(* CODESYS project ILG_Std_Lib
   Company: ILLIG packaging solutions
   DefaultNamespace: ILGStdLib
   Title: ILG_Std_Lib
   Version: 0.0.0.3

Project tree, tasks and I/O mapping:
  libraries: CXA_Utilities, 2.6.2.0 (Bosch Rexroth AG); CXA_CommonTypes, 3.4.0.0 (Bosch Rexroth AG); CXA_PLCopen, 3.4.0.3 (Bosch Rexroth AG); Standard, 3.5.18.0 (System); SysDir, 3.5.17.0 (System); SysFileAsync, 3.5.19.0 (System); SysTimeCore, 3.5.17.0 (System); SysTimeRtc, 3.5.20.0 (System); SysTypes, 3.1.2.0 (System); CXA_ctrlXIO, 1.20.11.0 (Bosch Rexroth AG); CXA_Datalayer, 3.4.0.0 (Bosch Rexroth AG); CXA_DriveUtil, 2.6.0.0 (Bosch Rexroth AG); CXA_FileAsync, 2.6.0.0 (Bosch Rexroth AG); CXA_Motion, 3.4.5.2 (Bosch Rexroth AG); CXA_MotionCore_fbs, 3.3.0.0 (Bosch Rexroth AG); CXA_MotionInterface, 3.4.0.3 (Bosch Rexroth AG); CXAC_Base, 1.18.4.0 (Bosch Rexroth AG); SysFile, 3.5.17.0 (System); File Access, 3.5.17.0 (3S - Smart Software Solutions GmbH); Software Engineering, 0.0.1 (Illig packaging solutions)
  libraries: CXA_Utilities, 2.6.2.0 (Bosch Rexroth AG); CXA_CommonTypes, 3.4.0.0 (Bosch Rexroth AG); CXA_PLCopen, 3.4.0.3 (Bosch Rexroth AG); Standard, 3.5.18.0 (System); SysDir, 3.5.17.0 (System); SysFileAsync, 3.5.19.0 (System); SysTimeCore, 3.5.17.0 (System); SysTimeRtc, 3.5.20.0 (System); SysTypes, 3.1.2.0 (System); CXA_ctrlXIO, 1.20.11.0 (Bosch Rexroth AG); CXA_Datalayer, 3.4.0.0 (Bosch Rexroth AG); CXA_DriveUtil, 2.6.0.0 (Bosch Rexroth AG); CXA_FileAsync, 2.6.0.0 (Bosch Rexroth AG); CXA_Motion, 3.4.5.2 (Bosch Rexroth AG); CXA_MotionCore_fbs, 3.3.0.0 (Bosch Rexroth AG); CXA_MotionInterface, 3.4.0.3 (Bosch Rexroth AG); CXAC_Base, 1.18.4.0 (Bosch Rexroth AG); SysFile, 3.5.17.0 (System); File Access, 3.5.17.0 (3S - Smart Software Solutions GmbH)
  00000000-0000-0000-0000-000000000000|D:\EIGENE_DATEIEN\GIT\libraries\SourceLibraries\CXA\CXA_Template\HistoryCXA_Template.txt
  0.7.0.0.Sync
  0.7.0.1.Sync
  _History/
    program _History_ [ST]
    History.txt
  _Library Informations/
    function GetLibVersion [ST]
    function GetLibVersionNumber [ST]
  commdata.all
  commdata.all
  commdata.all
  commdata.all
  Constants/
    GlobalKit/
      global variables GVL_ConstantsFlexProfile
      global variables GVL_ConstantsGlobalKit
  CXA_Library_Template.Sync
  function block FB_ArrayToWord_1 [ST]
  GeneralFunctionBlocks/
    ActivateDevices/
      Datatypes/
        ActConfig/
          data type ST_AxesActConfig
          data type ST_DeviceActConfig
          data type ST_DeviceActConfigBase
          data type ST_FirmwareType
          data type ST_InlineIOActConfig
          data type ST_ProfibusIOActConfig
          data type ST_SercosIOActConfig
          data type ST_SercosIOModuleActConfig
        CmdConfig/
          AxesConfig/
            data type ST_DoubleAxisConfig
            data type ST_FunctionalPackages
          data type ST_AxesCmdConfig
          data type ST_DeviceCmdConfig
          data type ST_DeviceCmdConfigBase
          data type ST_InlineIOCmdConfig
          data type ST_PNIOCmdConfig
          data type ST_PNIOModuleCmdConfig
          data type ST_ProfibusIOCmdConfig
          data type ST_SercosIOCmdConfig
          data type ST_SercosIOModuleCmdConfig
        data type E_InlineType
        data type E_S20Type
        Error/
          data type ST_AxesConfigError
          data type ST_AxesConfigErrorFoundDrives
          data type ST_DeviceConfigError
          data type ST_DeviceConfigErrorBase
          data type ST_InlineIOConfigError
          data type ST_ProfibusIOConfigError
          data type ST_SercosIOCmdConfigError
          data type ST_SercosIOConfigError
          data type ST_SercosIOModuleConfigError
        data type ST_DirEntry
        data type ST_SercosErrorReaction
      function block FB_ActivateDevices [ST]: _M_WriteLnString, M_0ReadActConfig, M_1ConfigAxes, M_2ConfigSercosIO, M_3ConfigInlineIO, M_4ConfigProfibsIO, M_5ConfigProfinetIO, M_8WriteConfig, M_9ErrorDone, M_DelStructure, M_Execute, M_GetSafetyType, M_GetSercosAdress, M_S20TypeToString, M_TypeCodeIsRexrothIO
      global variables GVL_ActivateDevices
      interface ITF_ActivateDevices: M_Execute
    ChangeNextDiagDelay/
      function block FB_ChangeNextDiagDelay [ST]
    function block FB_ArrayToWord [ST]
    function block FB_BlockAcknowledge10 [ST]
    function block FB_BlockAcknowledge21 [ST]
    function block FB_ClockMarker [ST]
    function block FB_Convert8BitTo5BitParameter [ST]
    function block FB_IlligOperatingModes [ST]
    function block FB_IlligZaehlstern [ST]
    function block FB_ParallelSteps [ST]
    function block FB_TimeBasedClockGenerator [ST]
    function block FB_TriggerValueChange [ST]
    function block FB_ValueIsIntegerMultiple [ST]
    function block FB_VIMP [ST]
  GeneralFunctions/
    Convert/
      function F_byWordToLeftByte [ST]
      function F_DwordToStrH5 [ST]
      function F_DwordToStrH8 [ST]
      function F_dwSwapDWordWord [ST]
      function F_iAnalogOutput4To20mA [ST]
      function F_rAnalogInput0To10V [ST]
      function F_rSwapReal [ST]
      function F_rSwapRealWord [ST]
      function F_Tad [ST]
      function F_WordToStrH [ST]
    ILG_Functions/
      function F_bCamDiscCalculation [ST]
      function F_InitArray [ST]
    Math/
      function F_lrRound [ST]
      function F_lrRoundRealToLReal [ST]
      function F_rModulo [ST]
      function F_rRound [ST]
      function F_rRoundGreater [ST]
      function F_rRoundTime [ST]
  Global Variables/
  ILG_Std_Lib.Sync
  ILG_Std_Lib.Sync
  ILG_Std_Lib.Sync
  ILG_Std_Lib.Sync
  InternalFunctions/
    function FUN_WriteLnString [ST]
  MachineDoorControllerInterface.Sync
  global variables ParaCxaLibraryTemplate
  program ReadMe [ST]
  Software Engineering.Sync
  Types/
    data type ST_Split
    data type T_CamTable
    data type T_ServoAxesArray
    data type T_Tables
  UnknownLibrary1.Sync
  UnknownLibrary21.Sync
  UnknownLibrary.Sync
*)

// Types/ST_Split
TYPE ST_Split :
STRUCT
	arWords:     ARRAY [1..400] OF POINTER TO STRING[255];
END_STRUCT
END_TYPE

// Types/T_CamTable
/// Ersetzt array vom Typ: ARRAY [1..99,1..1024] OF REAL; 
{attribute 'qualified_only' := ''}
{attribute 'namespace' := 'ILGStdLib.Types'}
TYPE T_CamTable :
ARRAY[1..99, 1..1024] OF REAL;
END_TYPE

// Types/T_ServoAxesArray
/// Ersetzt array vom Type: ARRAY[1..Max_Servoachsen, 0..Max_Segmente, 0..Max_Daten_pro_Segment] OF REAL
{attribute 'qualified_only' := ''}
{attribute 'namespace' := 'ILGStdLib.Types'}
TYPE T_ServoAxesArray :
ARRAY[1..GVL_ConstantsGlobalKit.iMAX_SERVO_AXES, 0..GVL_ConstantsGlobalKit.iMAX_SEGMENTS, 0..GVL_ConstantsGlobalKit.iMAX_DATA_PER_SEGMENT] OF REAL;
END_TYPE

// Types/T_Tables
/// Ersetzt array vom Type: ARRAY [1..Max_Anzahl_Stuetzpunkte, 1..Max_Anzahl_Tabellen] OF REAL; 
{attribute 'qualified_only' := ''}
{attribute 'namespace' := 'ILGStdLib.Types'}
TYPE T_Tables :
ARRAY[1..GVL_ConstantsGlobalKit.iMAX_COUNT_OF_SUPPORT_POINTS, 1..GVL_ConstantsGlobalKit.iMAX_COUNT_OF_TABLES] OF REAL;
END_TYPE

// GeneralFunctionBlocks/ActivateDevices/Datatypes/E_InlineType
{attribute 'qualified_only' := ''}
TYPE E_InlineType :
(
	///R-IB IL 24 DI 16-PAC 
	///R-IB IL 24 DI 16
	INLINE_DI16 := 16#BE01,
	///R-IB IL 24 DI 32/HD 
	///R-IB IL 24 DI 32/HD-PAC 
	///R-IB IL 24 DI 32/HD-NPN-PAC
	INLINE_DI32 := 16#BE02,
	///R-IB IL 24 DI 4
	///R-IB IL 24 DI 4-PAC
	///R-IB IL 24 EDI 2-DES
	///R-IB IL 24 DI 16-NPN-PAC 
	INLINE_DI4_2_16 := 16#BE41,
	///R-IB IL 24 DI 8
	///R-IB IL 24 DI 8-PAC
	INLINE_DI8 := 16#BE81,
	///R-IB IL 24 DI 2
	///R-IB IL 24 DI 2-PAC
	///R-IB IL 24 DI 2-NPN-PAC
	///IB IL 24 SEG/F-D-PAC
	INLINE_DI2_SEG := 16#BEC2,
	///R-IB IL 24 DO 16
	///R-IB IL 24 DO 16-PAC
	INLINE_DO16 := 16#BD01,
	///R-IB IL 24 DO 32/HD
	///R-IB IL 24 DO 32/HD-PAC
	///R-IB IL 24 DO 32/HD-NPN-PAC
	INLINE_DO32 := 16#BD02,
	///R-IB IL 24 DO 4
	///R-IB IL 24 DO 4-PAC
	///R-IB IL 24/230 DOR 4/W
	///R-IB IL 24/230 DOR 4/W-PAC
	INLINE_DO4_DOR4 := 16#BD41,
	///R-IB IL 24 DO 8
	///R-IB IL 24 DO 8-PAC
	///R-IB IL 24 DO 8-2A
	///R-IB IL 24 DO 8-2A-PAC
	///R-IB IL 24 DO 8-NPN-PAC
	INLINE_DO8 := 16#BD81,
	///R-IB IL 24 DO 2-2A
	///R-IB IL 24 DO 2-2A-PAC
	///R-IB IL 24 DO 2-NPN-PAC
	///R-IB IL 24/230 DOR 1/W
	///R-IB IL 24/230 DOR 1/W-PAC
	INLINE_DO2_DOR1 := 16#BDC2,
	///R-IB IL AI 8/SF-PAC
	///R-IB IL AI 8/IS-PAC
	INLINE_AI8 := 16#5F02,
	///R-IB IL AI 2/SF
	///R-IB IL AI 2/SF-PAC
	///R-IB IL AI 2/SF-230-PAC
	///R-IB IL TEMP 2 RTD
	///R-IB IL TEMP 2 RTD-PAC
	///R-IB IL TEMP 2 UTH-PAC
	///R-IB IL INC-IN-PAC
	INLINE_AI2_TEMP_INC_IN := 16#7F02,
	///R-IB IL SGI 2/F-PAC
	INLINE_SGI2 := 16#DF03,
	///R-IB IL AI 4/EF-PAC
	///R-IB IL TEMP 4/8 RTD-PAC
	INLINE_AI4_TEMP := 16#DF05,
	///R-IB IL AO 2/U/BP
	///R-IB IL AO 2/U/BP-PAC
	///R-IB IL AO 2/SF-PAC
	INLINE_AO2 := 16#5B02,
	///R-IB IL AO 1/SF
	///R-IB IL AO 1/SF-PAC
	INLINE_AO1 := 16#7D01,
	///R-IB IL CNT
	///R-IB IL CNT-PAC
	///R-IB IL INC-PAC
	///R-IB IL SSI-PAC
	///R-IB IL PWM/2-PAC
	///R-IB IL TEMPCON UTH-PAC
	INLINE_CNT_SSI_INC_PWM_TEMP := 16#BF02,
	///R-IL BK DDL
	INLINE_BK_DDL := 16#BF04,
	///R-IB IL RS232-PRO-PAC
	///R-IB IL RS485/422-PRO-PAC
	INLINE_RS232_RS485 := 16#BF06,
	///RF-FLM DI 8 M8
	INLINE_FLM_DI8 := 16#B281,
	///RF-FLM DIO 8/4 M8
	INLINE_FLM_DIO8 := 16#B381
);
END_TYPE

// GeneralFunctionBlocks/ActivateDevices/Datatypes/E_S20Type
{attribute 'qualified_only' := ''}
TYPE E_S20Type :
(
	///	undefinded
	S20_UNDEFINED := 16#0,
	///	S20-S3-BK+	Buskopf			R911173318
	S20_S3_BK_PLUS := 16#4158010099990002,
	///	S20-DI-16/4					R911172532
	S20_DI_16_4 := 16#41580002000000D0,
	///	S20-DO-16/3					R911172534
	S20_DO_16_3 := 16#41580002000000D1,
	///	S20-DI-32/1					R911172533
	S20_DI_32_1 := 16#41580004000000D2,
	///	S20-DO-32/1					R911172535
	S20_DO_32_1 := 16#41580004000000D3,
	///	S20-DO-8/2-2A				R911172541
	S20_DO_8_2_2A := 16#41580001000000D5,
	///	S20-DI-16/1					R911172543
	S20_DI_16_1 := 16#41580002000000D6,
	///	S20-DO-16/1					R911172542
	S20_DO_16_1 := 16#41580002000000D7,
	///	S20-AI-8					R911172536
	S20_AI_8 := 16#41580010000000A0,
	///	S20-AI-8-RTD				R911172537
	S20_AI_8_RTD := 16#41580010000000A1,
	///	S20-AI-8-UTH				R911172545               
	S20_AI_8_UTH := 16#41580012000000A2,
	///	S20-AO-8					R911172538
	S20_AO_8 := 16#41580010000000A3,
	///	S20-CNT-INC-2/2				R911172539
	S20_CNT_INC_2_2 := 16#4158001C000000F1,
	///	S20-SSI-AO-1/1				R911172544
	S20_SSI_AO_1_1 := 16#4158100C000000F2,
	///	Test_ChM					
	Placeholder_1 := 16#4158000400000008,
	///	Test_ChM					
	Placeholder_2 := 16#41580001000000D8,
	///	Test_ChM					
	Placeholder_3 := 16#4158000100000002,
	///	S20-AI-4-I					R911173249
	S20_AI_4_I := 16#41580008000000A6,
	///	S20-AI-4-U					R911173256
	S20_AI_4_U := 16#41580008000000A5,
	///	S20-DI-64/1					R911173340
	S20_DI_64_1 := 16#41580008000000D8,
	///	S20-DI-16/1-HS				R911173344
	S20_DI_16_1_HS := 16#41580002000000DB,
	///	S20-AI-4-RTD				R911173341
	S20_AI_4_RTD := 16#41580008000000A4,
	///	S20-RS-UNI					R911173343
	S20_RS_UNI := 16#41580814000000C0,
	///	S20-DIDO-8/1				R911173745               
	S20_DIDO_8_1 := 16#41580001000000DD,
	///	S20-AO-4					R911173248
	S20_AO_4 := 16#41580008000000A7,
	///	Test_ChM
	Placeholder_4 := 16#41580002000000DC,
	///	S20-AI-4-UTH				R911173342
	S20_AI_4_UTH := 16#41580008000000A8,
	///	SSDI-8/4					R911173191
	S20_SSDI_8_4 := 16#4158000A00000F00,
	///	SSDO-8/3					R911173192
	S20_SSDO_8_3 := 16#4158000A00000F01,
	///	S20-AI6-AO2-SSI2			R911173120
	S20_AI6_AO2_SSI2 := 16#41581014000000F3,
	///	S20-INC-2					R911173559
	S20_INC_2 := 16#41581014000000F5,
	///	S20-AIAO-2					R911173743
	S20_AIAO_2 := 16#41580008000000A9,
	///	S20-DO-64/1					R911173742
	S20_DO_64_1 := 16#41580008000000DF,
	///	S20-DOR-4/2-220-AC			R911173749
	S20_DOR_4_2_220_AC := 16#4158000100000D00,
	///	S20-DI-16/4-DO-8/3-HS		R911xxxxxx
	///  S20-SSI-AO-1_1				R911172544_AA1  fehlt in Buskoppler SDDML					
	S20_DI_16_4_DO_8_3_HS := 16#41580003010000D9
) LINT;
END_TYPE

// GeneralFunctionBlocks/ActivateDevices/Datatypes/ST_DirEntry
TYPE ST_DirEntry :
STRUCT
	sEntry: STRING;
	bDirectory: BOOL;
END_STRUCT
END_TYPE

// GeneralFunctionBlocks/ActivateDevices/Datatypes/ST_SercosErrorReaction
{attribute 'qualified_only' := ''}
{attribute 'strict' := ''}
TYPE ST_SercosErrorReaction :
STRUCT
	/// C-0-0506 Bit 0 = TRUE
	bF2Error: BOOL;
	/// C-0-0506 Bit 1 = TRUE
	bF5Error: BOOL;
	/// C-0-0506 Bit 0,1 = FALSE
	bF8Error: BOOL;
	/// Switch of E00B0179
	bNoRedundancyWarning: BOOL;
	bAutoRingRecovery: BOOL;
END_STRUCT
END_TYPE

// GeneralFunctionBlocks/ActivateDevices/Datatypes/ActConfig/ST_AxesActConfig
TYPE ST_AxesActConfig EXTENDS ST_DeviceActConfigBase :
STRUCT
	/// Name of Device 
	sName: STRING;
	/// TRUE = real Axis 
	bRealAxis: BOOL;
	/// TRUE = virtual Axis 
	bVirtualAxis: BOOL;
	/// Sercos address
	iSercosAddress: INT;
	/// Firmwarestring e.g. MPH-07 
	sFirmware: STRING;
	/// SNC or NOT 
	stFunctionalPackages: ST_FunctionalPackages;
	/// Which Axis of double Axis ? 
	stDoubleAxis: ST_DoubleAxisConfig;
	/// IP of drive S-0-1020
	sIP: STRING(16);
	/// serial no of Drive
	udiSerialNo: UDINT;
	/// String of SafetyType e.g. 'L3', 'S4', etc.	
	sSafetyType: STRING(2);
END_STRUCT
END_TYPE

// GeneralFunctionBlocks/ActivateDevices/Datatypes/ActConfig/ST_DeviceActConfig
TYPE ST_DeviceActConfig :
STRUCT
	astAxes: ARRAY[1..iMAX_AXES_NUMBER] OF ST_AxesActConfig;
	astSercosIO: ARRAY[1..iMAX_SERCOS_IO] OF ST_SercosIOActConfig;
	astInlineIO: ARRAY[1..iMAX_INLINE_IO] OF ST_InlineIOActConfig;
END_STRUCT
END_TYPE

// GeneralFunctionBlocks/ActivateDevices/Datatypes/ActConfig/ST_DeviceActConfigBase
TYPE ST_DeviceActConfigBase :
STRUCT
	/// TRUE = Device is present on the bus 
	bAvailable: BOOL;
END_STRUCT
END_TYPE

// GeneralFunctionBlocks/ActivateDevices/Datatypes/ActConfig/ST_FirmwareType
TYPE ST_FirmwareType :
STRUCT
	sType: STRING;
	iVersion: INT;
	iRelease: INT;
	bTestversion: BOOL;
END_STRUCT
END_TYPE

// GeneralFunctionBlocks/ActivateDevices/Datatypes/ActConfig/ST_InlineIOActConfig
TYPE ST_InlineIOActConfig EXTENDS ST_DeviceActConfigBase :
STRUCT
	eIOType: E_InlineType;
END_STRUCT
END_TYPE

// GeneralFunctionBlocks/ActivateDevices/Datatypes/ActConfig/ST_ProfibusIOActConfig
TYPE ST_ProfibusIOActConfig EXTENDS ST_DeviceActConfigBase :
STRUCT
END_STRUCT
END_TYPE

// GeneralFunctionBlocks/ActivateDevices/Datatypes/ActConfig/ST_SercosIOActConfig
TYPE ST_SercosIOActConfig EXTENDS ST_DeviceActConfigBase :
STRUCT
	/// Name of Device (will be taken from Cmd structure)
	sName: STRING;
	/// Sercos address
	iSercosAddress: INT;
	/// R911 TypeCode 
	sTypeCode: STRING;
	uiNoOfIO_Modules: UINT;
	astIOModule: ARRAY[0..GVL_ActivateDevices.iMAX_MODULE_ON_SERCOS_IO] OF ST_SercosIOModuleActConfig;
END_STRUCT
END_TYPE

// GeneralFunctionBlocks/ActivateDevices/Datatypes/ActConfig/ST_SercosIOModuleActConfig
TYPE ST_SercosIOModuleActConfig EXTENDS ST_DeviceActConfigBase :
STRUCT
	/// IO Module Type e.g. S20_DI_16_4
	IOType: E_S20Type;
END_STRUCT
END_TYPE

// GeneralFunctionBlocks/ActivateDevices/Datatypes/CmdConfig/ST_AxesCmdConfig
TYPE ST_AxesCmdConfig EXTENDS ST_DeviceCmdConfigBase :
STRUCT
	/// TRUE = real Axis 
	bRealAxis: BOOL;
	/// TRUE = virtual Axis 
	bVirtualAxis: BOOL;
	/// Sercos address
	iSercosAddress: INT;
	/// Firmwarestring e.g. MPH-07 
	sFirmware: STRING(8);
	/// SNC or NOT 
	stFunctionalPackages: ST_FunctionalPackages;
	/// String of SafetyType e.g. 'L3', 'S4', etc.
	sSafetyType: STRING(2);
	/// 	0: active, 
	///																						1: parked,
	///																						2: deactivated, 
	///																						4: active without command value processing,
	///																						5: parked with command value calculation,
	///																						6: deactivated with command value calculation 
	///																					
	iStatus: INT;
	/// Which Axis of double Axis ? 
	stDoubleAxis: ST_DoubleAxisConfig;
END_STRUCT
END_TYPE

// GeneralFunctionBlocks/ActivateDevices/Datatypes/CmdConfig/ST_DeviceCmdConfig
TYPE ST_DeviceCmdConfig :
STRUCT
	astAxes: ARRAY[1..iMAX_AXES_NUMBER] OF ST_AxesCmdConfig;
	astSercosIO: ARRAY[1..iMAX_SERCOS_IO] OF ST_SercosIOCmdConfig;
	astInlineIO: ARRAY[1..iMAX_INLINE_IO] OF ST_InlineIOCmdConfig;
	/// [x,0].Active = PROFINET MASTER is active
	astProfibusIO: ARRAY[1..iMAX_PROFIBUS_MASTER, 0..iMAX_PROFIBUS_SLAVE] OF ST_ProfibusIOCmdConfig;
	/// [x,0].Active = Profinet Master is active	(* 2020-07-06 gt: nach Vorlage "activateDevices_14.8.XM.iwz" von Jörg Schneider *)
	astPN_IO: ARRAY[1..iMAX_PN_MASTER, 0..iMAX_PN_SLAVE] OF ST_PNIOCmdConfig;
END_STRUCT
END_TYPE

// GeneralFunctionBlocks/ActivateDevices/Datatypes/CmdConfig/ST_DeviceCmdConfigBase
TYPE ST_DeviceCmdConfigBase :
STRUCT
	/// Name of Device 
	sName: STRING(80);
	/// TRUE = Device will be activated 
	bActive: BOOL;
END_STRUCT
END_TYPE

// GeneralFunctionBlocks/ActivateDevices/Datatypes/CmdConfig/ST_InlineIOCmdConfig
TYPE ST_InlineIOCmdConfig EXTENDS ST_DeviceCmdConfigBase :
STRUCT
	///IO is configured in IndraWorks	
	bConfigured: BOOL;
	/// which IO Type is used	 	
	eIOType: E_InlineType;
END_STRUCT
END_TYPE

// GeneralFunctionBlocks/ActivateDevices/Datatypes/CmdConfig/ST_PNIOCmdConfig
TYPE ST_PNIOCmdConfig EXTENDS ST_DeviceCmdConfigBase :
STRUCT
	///Fieldbus address 	
	sPNDeviceName: STRING(80);
	astIOModule: ARRAY[0..iMAX_MODULE_ON_PN_IO] OF ST_PNIOModuleCmdConfig;
END_STRUCT
END_TYPE

// GeneralFunctionBlocks/ActivateDevices/Datatypes/CmdConfig/ST_PNIOModuleCmdConfig
TYPE ST_PNIOModuleCmdConfig EXTENDS ST_DeviceCmdConfigBase :
STRUCT
	bConfigured: BOOL;
END_STRUCT
END_TYPE

// GeneralFunctionBlocks/ActivateDevices/Datatypes/CmdConfig/ST_ProfibusIOCmdConfig
TYPE ST_ProfibusIOCmdConfig EXTENDS ST_DeviceCmdConfigBase :
STRUCT
	///Fieldbus address
	iAddress: INT;
END_STRUCT
END_TYPE

// GeneralFunctionBlocks/ActivateDevices/Datatypes/CmdConfig/ST_SercosIOCmdConfig
TYPE ST_SercosIOCmdConfig EXTENDS ST_DeviceCmdConfigBase :
STRUCT
	/// Sercos address
	iSercosAddress: INT;
	///	Firmware 				:STRING;																(* Firmwarestring *)	
	astIOModule: ARRAY[0..iMAX_MODULE_ON_SERCOS_IO] OF ST_SercosIOModuleCmdConfig;
	/// will be calculated automatically if CheckSercosIOModuleConfig = TRUE
	uiNoOfIOModules: UINT;
END_STRUCT
END_TYPE

// GeneralFunctionBlocks/ActivateDevices/Datatypes/CmdConfig/ST_SercosIOModuleCmdConfig
TYPE ST_SercosIOModuleCmdConfig EXTENDS ST_DeviceCmdConfigBase :
STRUCT
	///IO Module is configured in IndraWorks		
	bConfigured: BOOL;
	/// IO Module Type e.g. S20_DI_16_4
	eIOType: E_S20Type;
END_STRUCT
END_TYPE

// GeneralFunctionBlocks/ActivateDevices/Datatypes/Error/ST_AxesConfigError
TYPE ST_AxesConfigError EXTENDS ST_DeviceConfigErrorBase :
STRUCT
	/// TRUE = Found drive has wrong SercosAddress
	bWrongSercosAddress: BOOL;
	/// TRUE = Found drive has wrong Firmware 
	bWrongFirmware: BOOL;
	/// TRUE = Found drive has wrong Functional Package
	bWrongFunctionalPackages: BOOL;
	/// TRUE = Found drive has wrong Doubleaxis Configuration
	bWrongDoubleAxisConfiguration: BOOL;
	/// TRUE = Found drive has wrong Safety option
	bWrongSafetyType: BOOL;
	/// TRUE = Drive is configured but not found
	bDriveConfiguredAndNotFound: BOOL;
	/// TRUE = Drive is found and configured in C-0-0478 (IndraWorks), but not configured at DeviceCmdConfig
	bDriveFoundAndNotConfigured: BOOL;
	/// Sercos Address of device 			
	iSercosAddress: INT;
END_STRUCT
END_TYPE

// GeneralFunctionBlocks/ActivateDevices/Datatypes/Error/ST_AxesConfigErrorFoundDrives
TYPE ST_AxesConfigErrorFoundDrives EXTENDS ST_DeviceConfigErrorBase :
STRUCT
	/// Sercos Address of device
	iSercosAddress: INT;
END_STRUCT
END_TYPE

// GeneralFunctionBlocks/ActivateDevices/Datatypes/Error/ST_DeviceConfigError
TYPE ST_DeviceConfigError :
STRUCT
	astAxes: ARRAY[1..iMAX_AXES_NUMBER] OF ST_AxesConfigError;
	///drive which were found but not configured in C-0-0478
	astFoundDrives: ARRAY[1..iMAX_AXES_NUMBER] OF ST_AxesConfigErrorFoundDrives;
	astSercosIO: ARRAY[1..iMAX_SERCOS_IO] OF ST_SercosIOConfigError;
	astInlineIO: ARRAY[1..iMAX_INLINE_IO] OF ST_InlineIOConfigError;
END_STRUCT
END_TYPE

// GeneralFunctionBlocks/ActivateDevices/Datatypes/Error/ST_DeviceConfigErrorBase
TYPE ST_DeviceConfigErrorBase :
STRUCT
	/// Name of Device (just for information)
	sName: STRING(80);
	/// TRUE = Error has been detected
	bError: BOOL;
	/// What is the Error?
	sErrorMessage: STRING(255);
END_STRUCT
END_TYPE

// GeneralFunctionBlocks/ActivateDevices/Datatypes/Error/ST_InlineIOConfigError
TYPE ST_InlineIOConfigError EXTENDS ST_DeviceConfigErrorBase :
STRUCT
	/// Wrong IO Type found or configured
	bWrongIOType: BOOL;
	/// TRUE = IO is configured but not found
	bIOConfiguredAndNotFound: BOOL;
	/// TRUE = IO is found but not configured in DeviceCmdConfig
	bIOFoundAndNotConfigured: BOOL;
END_STRUCT
END_TYPE

// GeneralFunctionBlocks/ActivateDevices/Datatypes/Error/ST_ProfibusIOConfigError
TYPE ST_ProfibusIOConfigError EXTENDS ST_DeviceConfigErrorBase :
STRUCT
END_STRUCT
END_TYPE

// GeneralFunctionBlocks/ActivateDevices/Datatypes/Error/ST_SercosIOCmdConfigError
TYPE ST_SercosIOCmdConfigError EXTENDS ST_DeviceConfigErrorBase :
STRUCT
	/// Too many IO configured in DeviceCmdConfig.sercos_IO
	bTooManyIOConfigured: BOOL;
	/// Too less IO configured in DeviceCmdConfig.sercos_IO
	bTooLessIOConfigured: BOOL;
	/// Sercos Address of device
	iSercosAddress: INT;
END_STRUCT
END_TYPE

// GeneralFunctionBlocks/ActivateDevices/Datatypes/Error/ST_SercosIOConfigError
TYPE ST_SercosIOConfigError EXTENDS ST_DeviceConfigErrorBase :
STRUCT
	/// TRUE = Found IO has wrong SercosAddress
	bWrongSercosAddress: BOOL;
	/// TRUE = IO is configured but not found
	bIOConfiguredAndNotFound: BOOL;
	/// TRUE = IO is found and configured in C-0-0478 (IndraWorks), but not configured at DeviceCmdConfig
	bIOFoundAndNotConfigured: BOOL;
	/// Sercos Address of device
	iSercosAddress: INT;
	astIO_Module: ARRAY[0..iMAX_MODULE_ON_SERCOS_IO] OF ST_SercosIOModuleConfigError;
	/// min one IO Module type is wrong	
	bWrongIOModuleType: BOOL;
	/// More IO Modules are configured in DeviceCmdConfig than found
	bMoreIOModulesConfiguredThanFound: BOOL;
	/// More IO Modules are found than configured in DeviceCmdConfig
	bMoreIOModulesFoundThanConfigured: BOOL;
END_STRUCT
END_TYPE

// GeneralFunctionBlocks/ActivateDevices/Datatypes/Error/ST_SercosIOModuleConfigError
TYPE ST_SercosIOModuleConfigError :
STRUCT
	/// TRUE = Found IOType is not equal to configured IOType
	bWrongIOType: BOOL;
END_STRUCT
END_TYPE

// GeneralFunctionBlocks/ActivateDevices/Datatypes/CmdConfig/AxesConfig/ST_DoubleAxisConfig
TYPE ST_DoubleAxisConfig :
STRUCT
	/// TRUE = Axis is part of double Axis 
	bIsDoubleAxis: BOOL;
	/// The sercos address of the left Axis 
	iLeftAxisAddress: INT;
	/// The sercos address of the right Axis 
	iRightAxisAddress: INT;
END_STRUCT
END_TYPE

// GeneralFunctionBlocks/ActivateDevices/Datatypes/CmdConfig/AxesConfig/ST_FunctionalPackages
TYPE ST_FunctionalPackages :
STRUCT
	bCl: BOOL := TRUE;
	bSnc: BOOL := FALSE;
	bSrv: BOOL := FALSE;
	bMsp: BOOL := FALSE;
	bTf: BOOL := FALSE;
	bMl: BOOL := FALSE;
	bMa: BOOL := FALSE;
END_STRUCT
END_TYPE

// ParaCxaLibraryTemplate
// These constants are editable by the user. After the value has been changed, an onlinechange is required.
// 
// .. note:: 
//   | If you want to change the values of these constants, this library may not be contained within the POUs. 
//   | The library has to be inserted below the device.
// 
// The effect of the pragma *{attribute ‘qualified_only’}* is that variables of a global variable list are only addressed BY specifying the global variable name, 
// for example array[ParaCxaLibraryTemplate.MIN_INDEX..ParaCxaLibraryTemplate.MAX_INDEX] OF BYTE




// Please adapt the name of the parameter list to the name of the library
{attribute ‘qualified_only’}
VAR_GLOBAL CONSTANT
    MIN_INDEX_:	UINT  :=  1;	(* Minimum index for arrays *)
    MAX_INDEX_:	UINT  :=  64;	(* Maximum number of elements *)
END_VAR

// Constants/GlobalKit/GVL_ConstantsFlexProfile
{attribute 'qualified_only' := ''}
{attribute 'namespace' := 'ILGStdLib.Consts.GVL_ConstantsFlexProfile'}
VAR_GLOBAL CONSTANT
	/// Speicherplatz Kurvenscheibentabelle 
	iCAM10_POL5_FAKT188_RIG: INT := 10;
	/// Speicherplatz Kurvenscheibentabelle 
	iCAM30_POL5_FAKT188_GIR: INT := 30;
	/// Speicherplatz Kurvenscheibentabelle 
	iCAM12_POL5_FAKT167_RIG: INT := 12;
	/// Speicherplatz Kurvenscheibentabelle 
	iCAM32_POL5_FAKT167_GIR: INT := 32;
	/// Speicherplatz Kurvenscheibentabelle 
	iCAM13_POL5_FAKT200_RIG: INT := 13;
	/// Speicherplatz Kurvenscheibentabelle 
	iCAM33_POL5_FAKT200_GIR: INT := 33;
	/// Speicherplatz Kurvenscheibentabelle 
	iCAM14_POL5_FAKT250_RIG: INT := 14;
	/// Speicherplatz Kurvenscheibentabelle 
	iCAM34_POL5_FAKT250_GIR: INT := 34;
	/// Speicherplatz Kurvenscheibentabelle 
	iCAM15_MOD_BE_TRA_RIG: INT := 15;
	/// Speicherplatz Kurvenscheibentabelle 
	iCAM35_MOD_BE_TRA_GIR: INT := 35;
	/// Speicherplatz Kurvenscheibentabelle 
	iCAM16_GEN_SINUS_RIG: INT := 16;
	/// Speicherplatz Kurvenscheibentabelle 
	iCAM36_GEN_SINUS_GIR: INT := 36;
	/// Speicherplatz Kurvenscheibentabelle 
	iCAM20_GIG: INT := 20;
	/// Speicherplatz Kurvenscheibentabelle 
	iCAM20_ZEIT: INT := 20;
	/// Speicherplatz Kurvenscheibentabelle 
	iCAM99_RIR: INT := 99;
END_VAR

// Constants/GlobalKit/GVL_ConstantsGlobalKit
{attribute 'qualified_only' := ''}
{attribute 'namespace' := 'ILGStdLib.Consts.GVL_ConstantsGlobalKit'}
VAR_GLOBAL CONSTANT
	/// Pi 
	rPI: REAL := 3.1415926535898;
	/// alt: Pi - Max. Anzahl der Servoachsen; Begrenzt druch die Anzahl der Spalten des Tabellenblatts 
	iMAX_SERVO_AXES: INT := 42;
	/// alt:  Max_Segmente - Max. Anzahl der Bewegungssegmente; begrenzt durch die Steuerung (2 Kurvenscheiben mit jeweils 16 Segmenten) 
	iMAX_SEGMENTS: INT := 32;
	/// alt: Max_Daten_pro_Segment - Max. Anzahl der Daten pro Bewegungssegment 
	iMAX_DATA_PER_SEGMENT: INT := 6;
	/// alt: Dezimalstellen_Zeit - Anzahl der Dezimalstellen der berechneten Zeiten 
	iDECIMALS_TIME: INT := 6;
	/// alt: Dezimalstellen_Weg - Anzahl der Dezimalstellen der berechneten Wege 
	iDECIMALS_WAY: INT := 6;
	/// alt: Dezimalstellen_Normierte_Profile - Anzahl der Dezimalstellen der normierten Profile 
	iDECIMALS_NORMALIZED_PROFILES: INT := 6;
	/// alt: Max_Anzahl_Stuetzpunkte_gk - Max. Anzahl der Stuetzpunkte eines Bewegungssegments 
	iMAX_COUNT_OF_SUPPORT_POINTS: INT := 1024;
	/// alt: Max_Anzahl_Tabellen - Max. Anzahl der Tabellen in der Steuerung 
	iMAX_COUNT_OF_TABLES: INT := 99;
END_VAR

// GeneralFunctionBlocks/ActivateDevices/GVL_ActivateDevices
///{attribute 'qualified_only'}
VAR_GLOBAL CONSTANT
	/// Maximum number of Axes depending on MLC type
	iMAX_AXES_NUMBER: INT := MB_MAX_AXIS_NUMBER;
	/// Maximum number of sercos IO (= MAX_SERCOS_DEVICES - actual no of Axes)
	iMAX_SERCOS_IO: INT := 20;
	/// Maximum number of Modules connected to sercos IO (Limit = 63)				
	iMAX_MODULE_ON_SERCOS_IO: INT := 32;
	/// Maximum number of Inline IO
	iMAX_INLINE_IO: INT := 20;
	/// Maximum number of S20 IO
	iMAX_S20_IO: INT := 20;
	/// Number of PROFIBUS Master Interfaces
	iMAX_PROFIBUS_MASTER: INT := 4;
	/// Number of PROFIBUS Slaves
	iMAX_PROFIBUS_SLAVE: INT := 10;
	/// Number of PROFINET Master Interfaces							(* 2020-07-06 gt: nach Vorlage "activateDevices_14.8.XM.iwz" von Jörg Schneider *)
	iMAX_PN_MASTER: INT := 4;
	/// Number of PROFINET Slaves									(* 2020-07-06 gt: nach Vorlage "activateDevices_14.8.XM.iwz" von Jörg Schneider *)
	iMAX_PN_SLAVE: INT := 10;
	/// Maximum number of Modules connected to PN IO (Limit = 63)	(* 2020-07-06 gt: nach Vorlage "activateDevices_14.8.XM.iwz" von Jörg Schneider *)
	iMAX_MODULE_ON_PN_IO: INT := 32;
	/// Maximum number of possible sercos devices
	iMAX_SERCOS_DEVICES: INT := MB_NUMBER_OF_SERCOS_DEVICES;
	/// Maximum number of lines in UserDefs.cfg
	iMAX_LINE_CFG: INT := 100;
	/// Maximum size for Buffervariable
	iMAX_BUFFER_SIZE: INT := (iMAX_LINE_CFG * 70);
	/// Maximum number of directory entrys
	iMAX_DIR_ENTRY: INT := 99;
	/// number of elements per device in C-0-0479
	iMAX_NUM_ELEMENTS_C479: INT := 9;
	/// number of elements per device in C-0-0578		
	iMAX_NUM_ELEMENTS_C578: INT := 8;
	/// Settings for CF filehandling
	sFILE_NAME: STRING := 'UserDefs.cfg';
	sPATH_NAME: STRING := '/ata0b';
	sFILE_AND_PATH: STRING := '/ata0b/UserDefs.cfg';
	///		stDriveFirmwarePath			: STRING := '/ata0b/DriveFirmware';
	/// Settings for MLC Diagnostic Logbook
	enSEVERITY: E_LOG_SEVERITY := E_LOG_SEVERITY.MESSAGE;
	enCLASS: E_LOG_CLASS := E_LOG_CLASS.CLASS_0;
	wDIAG_CODE: WORD := 16#0;
END_VAR

// FB_ArrayToWord_1
FUNCTION_BLOCK PUBLIC FB_ArrayToWord_1
(*####################################################################################################################################################
	
	Kurzbeschreibung:
		Funktionsbaustein zum Kopieren eines Arraybereichs in Variablen vom Datentyp WORD.

	Beschreibung:
		Am Eingang "iArray_Quelle_i" wird das zu kopierende Array parametriert. Über den Eingang "iStart_Offset_i" kann ein Offset 
		bezogen auf das am Eingang "iArray_Quelle_i" angegebene Array angegeben werden. Wird als "iStart_Offset_i" "0" angegeben so startet der 
		Kopiervorgang am ersten Feld des Eingang "iArray_Quelle_i".
		Der Eingang "iAnzahl_Worte_i" gibt die Anzahl der zu kopierende Worte bezogen auf den "iStart_Offset_i" an.
		An den Ausgängen "wZiel_Wort_1_o" ...."wZiel_Wort_16_o" können die Arrayinformationen Wortweise abgegriffen werden.
		
*******************************************************************************************************************************************************
	Historie:
		---------------------------------------------------------------------------------------------------------------------------------------------
		|	Datum			|		Name			|	Beschreibung																				|
		---------------------------------------------------------------------------------------------------------------------------------------------																						
		|	30.5.2011		|		T.Hauser		|	Baustein neu erstellt																		|
		---------------------------------------------------------------------------------------------------------------------------------------------
		|					|						|																								|
		---------------------------------------------------------------------------------------------------------------------------------------------
		|					|						|																								|
		---------------------------------------------------------------------------------------------------------------------------------------------
		|					|						|																								|
		---------------------------------------------------------------------------------------------------------------------------------------------

########################################################################################################################################################*)



(*******************************************************************************************************************************************)
(* Eingangsvariablen *)
(*******************************************************************************************************************************************)		
VAR_INPUT
	IN_pbArraySource:			POINTER TO BOOL;	(* Array aus dem der Datenbereich kopiert werden soll. Angabe ohne Index *)
	IN_bStartOffset:			BYTE; 				(* Defnition des ersten zu kopierenden Wert vom Eingang "iArray_Quelle_i" *)
	IN_bCountWords:				BYTE; 				(* Anzahl Worte die kopiert werden sollen*)
END_VAR

(*******************************************************************************************************************************************)
(* Ausgangsvariablen *)
(*******************************************************************************************************************************************)
VAR_OUTPUT
	OUT_wTargetWord1:				WORD;				(*Ziel Wort Bereich 1*)
	OUT_wTargetWord2:				WORD;				(*Ziel Wort Bereich 2*)
	OUT_wTargetWord3:				WORD;				(*Ziel Wort Bereich 3*)	
	OUT_wTargetWord4:				WORD;				(*Ziel Wort Bereich 4*)
	OUT_wTargetWord5:				WORD;				(*Ziel Wort Bereich 5*)
	OUT_wTargetWord6:				WORD;				(*Ziel Wort Bereich 6*)	
	OUT_wTargetWord7:				WORD;				(*Ziel Wort Bereich 7*)
	OUT_wTargetWord8:				WORD;				(*Ziel Wort Bereich 8*)
	OUT_wTargetWord9:				WORD;				(*Ziel Wort Bereich 9*)	
	OUT_wTargetWord10:				WORD;				(*Ziel Wort Bereich 10*)
	OUT_wTargetWord11:				WORD;				(*Ziel Wort Bereich 11*)
	OUT_wTargetWord12:				WORD;				(*Ziel Wort Bereich 12*)
	OUT_wTargetWord13:				WORD;				(*Ziel Wort Bereich 13*)	
	OUT_wTargetWord14:				WORD;				(*Ziel Wort Bereich 14*)
	OUT_wTargetWord15:				WORD;				(*Ziel Wort Bereich 15*)
	OUT_wTargetWord16:				WORD;				(*Ziel Wort Bereich 16*)
END_VAR

(*******************************************************************************************************************************************)
(* Interne Variablen *)
(*******************************************************************************************************************************************)
VAR
END_VAR

(* Anzahl der zu kopierenden Worte begrenzen *)
	IF IN_bCountWords > 16 THEN
		IN_bCountWords:= 16;
	END_IF

(* Startadresse vorbelegen*)
	IN_pbArraySource:= IN_pbArraySource + IN_bStartOffset;
(*******************************************************************************************************************************************)
(* Wort 1*)
(*******************************************************************************************************************************************)
(* Prüfen, ob Wort kopiert werden soll *)
	IF (IN_bCountWords >= 1) THEN
		(* Arraybereich kopieren *)
			OUT_wTargetWord1.0:=IN_pbArraySource^;
			IN_pbArraySource:=IN_pbArraySource+1;
			OUT_wTargetWord1.1:=IN_pbArraySource^;
			IN_pbArraySource:=IN_pbArraySource+1;
			OUT_wTargetWord1.2:=IN_pbArraySource^;
			IN_pbArraySource:=IN_pbArraySource+1;
			OUT_wTargetWord1.3:=IN_pbArraySource^;
			IN_pbArraySource:=IN_pbArraySource+1;
			OUT_wTargetWord1.4:=IN_pbArraySource^;
			IN_pbArraySource:=IN_pbArraySource+1;
			OUT_wTargetWord1.5:=IN_pbArraySource^;
			IN_pbArraySource:=IN_pbArraySource+1;
			OUT_wTargetWord1.6:=IN_pbArraySource^;
			IN_pbArraySource:=IN_pbArraySource+1;
			OUT_wTargetWord1.7:=IN_pbArraySource^;
			IN_pbArraySource:=IN_pbArraySource+1;
			OUT_wTargetWord1.8:=IN_pbArraySource^;
			IN_pbArraySource:=IN_pbArraySource+1;
			OUT_wTargetWord1.9:=IN_pbArraySource^;
			IN_pbArraySource:=IN_pbArraySource+1;
			OUT_wTargetWord1.10:=IN_pbArraySource^;
			IN_pbArraySource:=IN_pbArraySource+1;
			OUT_wTargetWord1.11:=IN_pbArraySource^;
			IN_pbArraySource:=IN_pbArraySource+1;
			OUT_wTargetWord1.12:=IN_pbArraySource^;
			IN_pbArraySource:=IN_pbArraySource+1;
			OUT_wTargetWord1.13:=IN_pbArraySource^;
			IN_pbArraySource:=IN_pbArraySource+1;
			OUT_wTargetWord1.14:=IN_pbArraySource^;
			IN_pbArraySource:=IN_pbArraySource+1;
			OUT_wTargetWord1.15:=IN_pbArraySource^;
			IN_pbArraySource:=IN_pbArraySource+1;
	END_IF

(*******************************************************************************************************************************************)
(* Wort 2*)
(*******************************************************************************************************************************************)
(* Prüfen, ob Wort kopiert werden soll *)
	IF (IN_bCountWords >= 2) THEN
		(* Arraybereich kopieren *)
			OUT_wTargetWord2.0:=IN_pbArraySource^;
			IN_pbArraySource:=IN_pbArraySource+1;
			OUT_wTargetWord2.1:=IN_pbArraySource^;
			IN_pbArraySource:=IN_pbArraySource+1;
			OUT_wTargetWord2.2:=IN_pbArraySource^;
			IN_pbArraySource:=IN_pbArraySource+1;
			OUT_wTargetWord2.3:=IN_pbArraySource^;
			IN_pbArraySource:=IN_pbArraySource+1;
			OUT_wTargetWord2.4:=IN_pbArraySource^;
			IN_pbArraySource:=IN_pbArraySource+1;
			OUT_wTargetWord2.5:=IN_pbArraySource^;
			IN_pbArraySource:=IN_pbArraySource+1;
			OUT_wTargetWord2.6:=IN_pbArraySource^;
			IN_pbArraySource:=IN_pbArraySource+1;
			OUT_wTargetWord2.7:=IN_pbArraySource^;
			IN_pbArraySource:=IN_pbArraySource+1;
			OUT_wTargetWord2.8:=IN_pbArraySource^;
			IN_pbArraySource:=IN_pbArraySource+1;
			OUT_wTargetWord2.9:=IN_pbArraySource^;
			IN_pbArraySource:=IN_pbArraySource+1;
			OUT_wTargetWord2.10:=IN_pbArraySource^;
			IN_pbArraySource:=IN_pbArraySource+1;
			OUT_wTargetWord2.11:=IN_pbArraySource^;
			IN_pbArraySource:=IN_pbArraySource+1;
			OUT_wTargetWord2.12:=IN_pbArraySource^;
			IN_pbArraySource:=IN_pbArraySource+1;
			OUT_wTargetWord2.13:=IN_pbArraySource^;
			IN_pbArraySource:=IN_pbArraySource+1;
			OUT_wTargetWord2.14:=IN_pbArraySource^;
			IN_pbArraySource:=IN_pbArraySource+1;
			OUT_wTargetWord2.15:=IN_pbArraySource^;
			IN_pbArraySource:=IN_pbArraySource+1;
	END_IF		
		
(*******************************************************************************************************************************************)
(* Wort 3*)
(*******************************************************************************************************************************************)
(* Prüfen, ob Wort kopiert werden soll *)
	IF (IN_bCountWords >= 3) THEN
	(* Arraybereich kopieren *)
		OUT_wTargetWord3.0:=IN_pbArraySource^;
		IN_pbArraySource:=IN_pbArraySource+1;
		OUT_wTargetWord3.1:=IN_pbArraySource^;
		IN_pbArraySource:=IN_pbArraySource+1;
		OUT_wTargetWord3.2:=IN_pbArraySource^;
		IN_pbArraySource:=IN_pbArraySource+1;
		OUT_wTargetWord3.3:=IN_pbArraySource^;
		IN_pbArraySource:=IN_pbArraySource+1;
		OUT_wTargetWord3.4:=IN_pbArraySource^;
		IN_pbArraySource:=IN_pbArraySource+1;
		OUT_wTargetWord3.5:=IN_pbArraySource^;
		IN_pbArraySource:=IN_pbArraySource+1;
		OUT_wTargetWord3.6:=IN_pbArraySource^;
		IN_pbArraySource:=IN_pbArraySource+1;
		OUT_wTargetWord3.7:=IN_pbArraySource^;
		IN_pbArraySource:=IN_pbArraySource+1;
		OUT_wTargetWord3.8:=IN_pbArraySource^;
		IN_pbArraySource:=IN_pbArraySource+1;
		OUT_wTargetWord3.9:=IN_pbArraySource^;
		IN_pbArraySource:=IN_pbArraySource+1;
		OUT_wTargetWord3.10:=IN_pbArraySource^;
		IN_pbArraySource:=IN_pbArraySource+1;
		OUT_wTargetWord3.11:=IN_pbArraySource^;
		IN_pbArraySource:=IN_pbArraySource+1;
		OUT_wTargetWord3.12:=IN_pbArraySource^;
		IN_pbArraySource:=IN_pbArraySource+1;
		OUT_wTargetWord3.13:=IN_pbArraySource^;
		IN_pbArraySource:=IN_pbArraySource+1;
		OUT_wTargetWord3.14:=IN_pbArraySource^;
		IN_pbArraySource:=IN_pbArraySource+1;
		OUT_wTargetWord3.15:=IN_pbArraySource^;
		IN_pbArraySource:=IN_pbArraySource+1;
	END_IF		
	
(*******************************************************************************************************************************************)
(* Wort 4*)
(*******************************************************************************************************************************************)
(* Prüfen, ob Wort kopiert werden soll *)
	IF (IN_bCountWords >= 4) THEN
	(* Arraybereich kopieren *)
		OUT_wTargetWord4.0:=IN_pbArraySource^;
		IN_pbArraySource:=IN_pbArraySource+1;
		OUT_wTargetWord4.1:=IN_pbArraySource^;
		IN_pbArraySource:=IN_pbArraySource+1;
		OUT_wTargetWord4.2:=IN_pbArraySource^;
		IN_pbArraySource:=IN_pbArraySource+1;
		OUT_wTargetWord4.3:=IN_pbArraySource^;
		IN_pbArraySource:=IN_pbArraySource+1;
		OUT_wTargetWord4.4:=IN_pbArraySource^;
		IN_pbArraySource:=IN_pbArraySource+1;
		OUT_wTargetWord4.5:=IN_pbArraySource^;
		IN_pbArraySource:=IN_pbArraySource+1;
		OUT_wTargetWord4.6:=IN_pbArraySource^;
		IN_pbArraySource:=IN_pbArraySource+1;
		OUT_wTargetWord4.7:=IN_pbArraySource^;
		IN_pbArraySource:=IN_pbArraySource+1;
		OUT_wTargetWord4.8:=IN_pbArraySource^;
		IN_pbArraySource:=IN_pbArraySource+1;
		OUT_wTargetWord4.9:=IN_pbArraySource^;
		IN_pbArraySource:=IN_pbArraySource+1;
		OUT_wTargetWord4.10:=IN_pbArraySource^;
		IN_pbArraySource:=IN_pbArraySource+1;
		OUT_wTargetWord4.11:=IN_pbArraySource^;
		IN_pbArraySource:=IN_pbArraySource+1;
		OUT_wTargetWord4.12:=IN_pbArraySource^;
		IN_pbArraySource:=IN_pbArraySource+1;
		OUT_wTargetWord4.13:=IN_pbArraySource^;
		IN_pbArraySource:=IN_pbArraySource+1;
		OUT_wTargetWord4.14:=IN_pbArraySource^;
		IN_pbArraySource:=IN_pbArraySource+1;
		OUT_wTargetWord4.15:=IN_pbArraySource^;
		IN_pbArraySource:=IN_pbArraySource+1;
	END_IF			

(*******************************************************************************************************************************************)
(* Wort 5*)
(*******************************************************************************************************************************************)
(* Prüfen, ob Wort kopiert werden soll *)
	IF (IN_bCountWords >= 5) THEN
	(* Arraybereich kopieren *)
		OUT_wTargetWord5.0:=IN_pbArraySource^;
		IN_pbArraySource:=IN_pbArraySource+1;
		OUT_wTargetWord5.1:=IN_pbArraySource^;
		IN_pbArraySource:=IN_pbArraySource+1;
		OUT_wTargetWord5.2:=IN_pbArraySource^;
		IN_pbArraySource:=IN_pbArraySource+1;
		OUT_wTargetWord5.3:=IN_pbArraySource^;
		IN_pbArraySource:=IN_pbArraySource+1;
		OUT_wTargetWord5.4:=IN_pbArraySource^;
		IN_pbArraySource:=IN_pbArraySource+1;
		OUT_wTargetWord5.5:=IN_pbArraySource^;
		IN_pbArraySource:=IN_pbArraySource+1;
		OUT_wTargetWord5.6:=IN_pbArraySource^;
		IN_pbArraySource:=IN_pbArraySource+1;
		OUT_wTargetWord5.7:=IN_pbArraySource^;
		IN_pbArraySource:=IN_pbArraySource+1;
		OUT_wTargetWord5.8:=IN_pbArraySource^;
		IN_pbArraySource:=IN_pbArraySource+1;
		OUT_wTargetWord5.9:=IN_pbArraySource^;
		IN_pbArraySource:=IN_pbArraySource+1;
		OUT_wTargetWord5.10:=IN_pbArraySource^;
		IN_pbArraySource:=IN_pbArraySource+1;
		OUT_wTargetWord5.11:=IN_pbArraySource^;
		IN_pbArraySource:=IN_pbArraySource+1;
		OUT_wTargetWord5.12:=IN_pbArraySource^;
		IN_pbArraySource:=IN_pbArraySource+1;
		OUT_wTargetWord5.13:=IN_pbArraySource^;
		IN_pbArraySource:=IN_pbArraySource+1;
		OUT_wTargetWord5.14:=IN_pbArraySource^;
		IN_pbArraySource:=IN_pbArraySource+1;
		OUT_wTargetWord5.15:=IN_pbArraySource^;
		IN_pbArraySource:=IN_pbArraySource+1;
	END_IF			

(*******************************************************************************************************************************************)
(* Wort 6*)
(*******************************************************************************************************************************************)
(* Prüfen, ob Wort kopiert werden soll *)
	IF (IN_bCountWords >= 6) THEN
	(* Arraybereich kopieren *)
		OUT_wTargetWord6.0:=IN_pbArraySource^;
		IN_pbArraySource:=IN_pbArraySource+1;
		OUT_wTargetWord6.1:=IN_pbArraySource^;
		IN_pbArraySource:=IN_pbArraySource+1;
		OUT_wTargetWord6.2:=IN_pbArraySource^;
		IN_pbArraySource:=IN_pbArraySource+1;
		OUT_wTargetWord6.3:=IN_pbArraySource^;
		IN_pbArraySource:=IN_pbArraySource+1;
		OUT_wTargetWord6.4:=IN_pbArraySource^;
		IN_pbArraySource:=IN_pbArraySource+1;
		OUT_wTargetWord6.5:=IN_pbArraySource^;
		IN_pbArraySource:=IN_pbArraySource+1;
		OUT_wTargetWord6.6:=IN_pbArraySource^;
		IN_pbArraySource:=IN_pbArraySource+1;
		OUT_wTargetWord6.7:=IN_pbArraySource^;
		IN_pbArraySource:=IN_pbArraySource+1;
		OUT_wTargetWord6.8:=IN_pbArraySource^;
		IN_pbArraySource:=IN_pbArraySource+1;
		OUT_wTargetWord6.9:=IN_pbArraySource^;
		IN_pbArraySource:=IN_pbArraySource+1;
		OUT_wTargetWord6.10:=IN_pbArraySource^;
		IN_pbArraySource:=IN_pbArraySource+1;
		OUT_wTargetWord6.11:=IN_pbArraySource^;
		IN_pbArraySource:=IN_pbArraySource+1;
		OUT_wTargetWord6.12:=IN_pbArraySource^;
		IN_pbArraySource:=IN_pbArraySource+1;
		OUT_wTargetWord6.13:=IN_pbArraySource^;
		IN_pbArraySource:=IN_pbArraySource+1;
		OUT_wTargetWord6.14:=IN_pbArraySource^;
		IN_pbArraySource:=IN_pbArraySource+1;
		OUT_wTargetWord6.15:=IN_pbArraySource^;
		IN_pbArraySource:=IN_pbArraySource+1;
END_IF
		
(*******************************************************************************************************************************************)
(* Wort 7*)
(*******************************************************************************************************************************************)
(* Prüfen, ob Wort kopiert werden soll *)
	IF (IN_bCountWords >= 7) THEN
	(* Arraybereich kopieren *)
		OUT_wTargetWord7.0:=IN_pbArraySource^;
		IN_pbArraySource:=IN_pbArraySource+1;
		OUT_wTargetWord7.1:=IN_pbArraySource^;
		IN_pbArraySource:=IN_pbArraySource+1;
		OUT_wTargetWord7.2:=IN_pbArraySource^;
		IN_pbArraySource:=IN_pbArraySource+1;
		OUT_wTargetWord7.3:=IN_pbArraySource^;
		IN_pbArraySource:=IN_pbArraySource+1;
		OUT_wTargetWord7.4:=IN_pbArraySource^;
		IN_pbArraySource:=IN_pbArraySource+1;
		OUT_wTargetWord7.5:=IN_pbArraySource^;
		IN_pbArraySource:=IN_pbArraySource+1;
		OUT_wTargetWord7.6:=IN_pbArraySource^;
		IN_pbArraySource:=IN_pbArraySource+1;
		OUT_wTargetWord7.7:=IN_pbArraySource^;
		IN_pbArraySource:=IN_pbArraySource+1;
		OUT_wTargetWord7.8:=IN_pbArraySource^;
		IN_pbArraySource:=IN_pbArraySource+1;
		OUT_wTargetWord7.9:=IN_pbArraySource^;
		IN_pbArraySource:=IN_pbArraySource+1;
		OUT_wTargetWord7.10:=IN_pbArraySource^;
		IN_pbArraySource:=IN_pbArraySource+1;
		OUT_wTargetWord7.11:=IN_pbArraySource^;
		IN_pbArraySource:=IN_pbArraySource+1;
		OUT_wTargetWord7.12:=IN_pbArraySource^;
		IN_pbArraySource:=IN_pbArraySource+1;
		OUT_wTargetWord7.13:=IN_pbArraySource^;
		IN_pbArraySource:=IN_pbArraySource+1;
		OUT_wTargetWord7.14:=IN_pbArraySource^;
		IN_pbArraySource:=IN_pbArraySource+1;
		OUT_wTargetWord7.15:=IN_pbArraySource^;
		IN_pbArraySource:=IN_pbArraySource+1;
	END_IF	
		
(*******************************************************************************************************************************************)
(* Wort 8*)
(*******************************************************************************************************************************************)
(* Prüfen, ob Wort kopiert werden soll *)
	IF (IN_bCountWords >= 8) THEN
	(* Arraybereich kopieren *)
		OUT_wTargetWord8.0:=IN_pbArraySource^;
		IN_pbArraySource:=IN_pbArraySource+1;
		OUT_wTargetWord8.1:=IN_pbArraySource^;
		IN_pbArraySource:=IN_pbArraySource+1;
		OUT_wTargetWord8.2:=IN_pbArraySource^;
		IN_pbArraySource:=IN_pbArraySource+1;
		OUT_wTargetWord8.3:=IN_pbArraySource^;
		IN_pbArraySource:=IN_pbArraySource+1;
		OUT_wTargetWord8.4:=IN_pbArraySource^;
		IN_pbArraySource:=IN_pbArraySource+1;
		OUT_wTargetWord8.5:=IN_pbArraySource^;
		IN_pbArraySource:=IN_pbArraySource+1;
		OUT_wTargetWord8.6:=IN_pbArraySource^;
		IN_pbArraySource:=IN_pbArraySource+1;
		OUT_wTargetWord8.7:=IN_pbArraySource^;
		IN_pbArraySource:=IN_pbArraySource+1;
		OUT_wTargetWord8.8:=IN_pbArraySource^;
		IN_pbArraySource:=IN_pbArraySource+1;
		OUT_wTargetWord8.9:=IN_pbArraySource^;
		IN_pbArraySource:=IN_pbArraySource+1;
		OUT_wTargetWord8.10:=IN_pbArraySource^;
		IN_pbArraySource:=IN_pbArraySource+1;
		OUT_wTargetWord8.11:=IN_pbArraySource^;
		IN_pbArraySource:=IN_pbArraySource+1;
		OUT_wTargetWord8.12:=IN_pbArraySource^;
		IN_pbArraySource:=IN_pbArraySource+1;
		OUT_wTargetWord8.13:=IN_pbArraySource^;
		IN_pbArraySource:=IN_pbArraySource+1;
		OUT_wTargetWord8.14:=IN_pbArraySource^;
		IN_pbArraySource:=IN_pbArraySource+1;
		OUT_wTargetWord8.15:=IN_pbArraySource^;
		IN_pbArraySource:=IN_pbArraySource+1;
	END_IF	

(*******************************************************************************************************************************************)
(* Wort 9*)
(*******************************************************************************************************************************************)
(* Prüfen, ob Wort kopiert werden soll *)
	IF (IN_bCountWords >= 9) THEN
	(* Arraybereich kopieren *)
		OUT_wTargetWord9.0:=IN_pbArraySource^;
		IN_pbArraySource:=IN_pbArraySource+1;
		OUT_wTargetWord9.1:=IN_pbArraySource^;
		IN_pbArraySource:=IN_pbArraySource+1;
		OUT_wTargetWord9.2:=IN_pbArraySource^;
		IN_pbArraySource:=IN_pbArraySource+1;
		OUT_wTargetWord9.3:=IN_pbArraySource^;
		IN_pbArraySource:=IN_pbArraySource+1;
		OUT_wTargetWord9.4:=IN_pbArraySource^;
		IN_pbArraySource:=IN_pbArraySource+1;
		OUT_wTargetWord9.5:=IN_pbArraySource^;
		IN_pbArraySource:=IN_pbArraySource+1;
		OUT_wTargetWord9.6:=IN_pbArraySource^;
		IN_pbArraySource:=IN_pbArraySource+1;
		OUT_wTargetWord9.7:=IN_pbArraySource^;
		IN_pbArraySource:=IN_pbArraySource+1;
		OUT_wTargetWord9.8:=IN_pbArraySource^;
		IN_pbArraySource:=IN_pbArraySource+1;
		OUT_wTargetWord9.9:=IN_pbArraySource^;
		IN_pbArraySource:=IN_pbArraySource+1;
		OUT_wTargetWord9.10:=IN_pbArraySource^;
		IN_pbArraySource:=IN_pbArraySource+1;
		OUT_wTargetWord9.11:=IN_pbArraySource^;
		IN_pbArraySource:=IN_pbArraySource+1;
		OUT_wTargetWord9.12:=IN_pbArraySource^;
		IN_pbArraySource:=IN_pbArraySource+1;
		OUT_wTargetWord9.13:=IN_pbArraySource^;
		IN_pbArraySource:=IN_pbArraySource+1;
		OUT_wTargetWord9.14:=IN_pbArraySource^;
		IN_pbArraySource:=IN_pbArraySource+1;
		OUT_wTargetWord9.15:=IN_pbArraySource^;
		IN_pbArraySource:=IN_pbArraySource+1;
	END_IF	

(*******************************************************************************************************************************************)
(* Wort 10*)
(*******************************************************************************************************************************************)
(* Prüfen, ob Wort kopiert werden soll *)
	IF (IN_bCountWords >= 10) THEN
	(* Arraybereich kopieren *)
		OUT_wTargetWord10.0:=IN_pbArraySource^;
		IN_pbArraySource:=IN_pbArraySource+1;
		OUT_wTargetWord10.1:=IN_pbArraySource^;
		IN_pbArraySource:=IN_pbArraySource+1;
		OUT_wTargetWord10.2:=IN_pbArraySource^;
		IN_pbArraySource:=IN_pbArraySource+1;
		OUT_wTargetWord10.3:=IN_pbArraySource^;
		IN_pbArraySource:=IN_pbArraySource+1;
		OUT_wTargetWord10.4:=IN_pbArraySource^;
		IN_pbArraySource:=IN_pbArraySource+1;
		OUT_wTargetWord10.5:=IN_pbArraySource^;
		IN_pbArraySource:=IN_pbArraySource+1;
		OUT_wTargetWord10.6:=IN_pbArraySource^;
		IN_pbArraySource:=IN_pbArraySource+1;
		OUT_wTargetWord10.7:=IN_pbArraySource^;
		IN_pbArraySource:=IN_pbArraySource+1;
		OUT_wTargetWord10.8:=IN_pbArraySource^;
		IN_pbArraySource:=IN_pbArraySource+1;
		OUT_wTargetWord10.9:=IN_pbArraySource^;
		IN_pbArraySource:=IN_pbArraySource+1;
		OUT_wTargetWord10.10:=IN_pbArraySource^;
		IN_pbArraySource:=IN_pbArraySource+1;
		OUT_wTargetWord10.11:=IN_pbArraySource^;
		IN_pbArraySource:=IN_pbArraySource+1;
		OUT_wTargetWord10.12:=IN_pbArraySource^;
		IN_pbArraySource:=IN_pbArraySource+1;
		OUT_wTargetWord10.13:=IN_pbArraySource^;
		IN_pbArraySource:=IN_pbArraySource+1;
		OUT_wTargetWord10.14:=IN_pbArraySource^;
		IN_pbArraySource:=IN_pbArraySource+1;
		OUT_wTargetWord10.15:=IN_pbArraySource^;
		IN_pbArraySource:=IN_pbArraySource+1;
	END_IF		

(*******************************************************************************************************************************************)
(* Wort 11*)
(*******************************************************************************************************************************************)
(* Prüfen, ob Wort kopiert werden soll *)
	IF (IN_bCountWords >= 11) THEN
	(* Arraybereich kopieren *)
		OUT_wTargetWord11.0:=IN_pbArraySource^;
		IN_pbArraySource:=IN_pbArraySource+1;
		OUT_wTargetWord11.1:=IN_pbArraySource^;
		IN_pbArraySource:=IN_pbArraySource+1;
		OUT_wTargetWord11.2:=IN_pbArraySource^;
		IN_pbArraySource:=IN_pbArraySource+1;
		OUT_wTargetWord11.3:=IN_pbArraySource^;
		IN_pbArraySource:=IN_pbArraySource+1;
		OUT_wTargetWord11.4:=IN_pbArraySource^;
		IN_pbArraySource:=IN_pbArraySource+1;
		OUT_wTargetWord11.5:=IN_pbArraySource^;
		IN_pbArraySource:=IN_pbArraySource+1;
		OUT_wTargetWord11.6:=IN_pbArraySource^;
		IN_pbArraySource:=IN_pbArraySource+1;
		OUT_wTargetWord11.7:=IN_pbArraySource^;
		IN_pbArraySource:=IN_pbArraySource+1;
		OUT_wTargetWord11.8:=IN_pbArraySource^;
		IN_pbArraySource:=IN_pbArraySource+1;
		OUT_wTargetWord11.9:=IN_pbArraySource^;
		IN_pbArraySource:=IN_pbArraySource+1;
		OUT_wTargetWord11.10:=IN_pbArraySource^;
		IN_pbArraySource:=IN_pbArraySource+1;
		OUT_wTargetWord11.11:=IN_pbArraySource^;
		IN_pbArraySource:=IN_pbArraySource+1;
		OUT_wTargetWord11.12:=IN_pbArraySource^;
		IN_pbArraySource:=IN_pbArraySource+1;
		OUT_wTargetWord11.13:=IN_pbArraySource^;
		IN_pbArraySource:=IN_pbArraySource+1;
		OUT_wTargetWord11.14:=IN_pbArraySource^;
		IN_pbArraySource:=IN_pbArraySource+1;
		OUT_wTargetWord11.15:=IN_pbArraySource^;
		IN_pbArraySource:=IN_pbArraySource+1;
	END_IF		
	
(*******************************************************************************************************************************************)
(* Wort 12*)
(*******************************************************************************************************************************************)
(* Prüfen, ob Wort kopiert werden soll *)
	IF (IN_bCountWords >= 12) THEN
	(* Arraybereich kopieren *)
		OUT_wTargetWord12.0:=IN_pbArraySource^;
		IN_pbArraySource:=IN_pbArraySource+1;
		OUT_wTargetWord12.1:=IN_pbArraySource^;
		IN_pbArraySource:=IN_pbArraySource+1;
		OUT_wTargetWord12.2:=IN_pbArraySource^;
		IN_pbArraySource:=IN_pbArraySource+1;
		OUT_wTargetWord12.3:=IN_pbArraySource^;
		IN_pbArraySource:=IN_pbArraySource+1;
		OUT_wTargetWord12.4:=IN_pbArraySource^;
		IN_pbArraySource:=IN_pbArraySource+1;
		OUT_wTargetWord12.5:=IN_pbArraySource^;
		IN_pbArraySource:=IN_pbArraySource+1;
		OUT_wTargetWord12.6:=IN_pbArraySource^;
		IN_pbArraySource:=IN_pbArraySource+1;
		OUT_wTargetWord12.7:=IN_pbArraySource^;
		IN_pbArraySource:=IN_pbArraySource+1;
		OUT_wTargetWord12.8:=IN_pbArraySource^;
		IN_pbArraySource:=IN_pbArraySource+1;
		OUT_wTargetWord12.9:=IN_pbArraySource^;
		IN_pbArraySource:=IN_pbArraySource+1;
		OUT_wTargetWord12.10:=IN_pbArraySource^;
		IN_pbArraySource:=IN_pbArraySource+1;
		OUT_wTargetWord12.11:=IN_pbArraySource^;
		IN_pbArraySource:=IN_pbArraySource+1;
		OUT_wTargetWord12.12:=IN_pbArraySource^;
		IN_pbArraySource:=IN_pbArraySource+1;
		OUT_wTargetWord12.13:=IN_pbArraySource^;
		IN_pbArraySource:=IN_pbArraySource+1;
		OUT_wTargetWord12.14:=IN_pbArraySource^;
		IN_pbArraySource:=IN_pbArraySource+1;
		OUT_wTargetWord12.15:=IN_pbArraySource^;
		IN_pbArraySource:=IN_pbArraySource+1;
	END_IF	

(*******************************************************************************************************************************************)
(* Wort 13*)
(*******************************************************************************************************************************************)
(* Prüfen, ob Wort kopiert werden soll *)
	IF (IN_bCountWords >= 13) THEN
	(* Arraybereich kopieren *)
		OUT_wTargetWord13.0:=IN_pbArraySource^;
		IN_pbArraySource:=IN_pbArraySource+1;
		OUT_wTargetWord13.1:=IN_pbArraySource^;
		IN_pbArraySource:=IN_pbArraySource+1;
		OUT_wTargetWord13.2:=IN_pbArraySource^;
		IN_pbArraySource:=IN_pbArraySource+1;
		OUT_wTargetWord13.3:=IN_pbArraySource^;
		IN_pbArraySource:=IN_pbArraySource+1;
		OUT_wTargetWord13.4:=IN_pbArraySource^;
		IN_pbArraySource:=IN_pbArraySource+1;
		OUT_wTargetWord13.5:=IN_pbArraySource^;
		IN_pbArraySource:=IN_pbArraySource+1;
		OUT_wTargetWord13.6:=IN_pbArraySource^;
		IN_pbArraySource:=IN_pbArraySource+1;
		OUT_wTargetWord13.7:=IN_pbArraySource^;
		IN_pbArraySource:=IN_pbArraySource+1;
		OUT_wTargetWord13.8:=IN_pbArraySource^;
		IN_pbArraySource:=IN_pbArraySource+1;
		OUT_wTargetWord13.9:=IN_pbArraySource^;
		IN_pbArraySource:=IN_pbArraySource+1;
		OUT_wTargetWord13.10:=IN_pbArraySource^;
		IN_pbArraySource:=IN_pbArraySource+1;
		OUT_wTargetWord13.11:=IN_pbArraySource^;
		IN_pbArraySource:=IN_pbArraySource+1;
		OUT_wTargetWord13.12:=IN_pbArraySource^;
		IN_pbArraySource:=IN_pbArraySource+1;
		OUT_wTargetWord13.13:=IN_pbArraySource^;
		IN_pbArraySource:=IN_pbArraySource+1;
		OUT_wTargetWord13.14:=IN_pbArraySource^;
		IN_pbArraySource:=IN_pbArraySource+1;
		OUT_wTargetWord13.15:=IN_pbArraySource^;
		IN_pbArraySource:=IN_pbArraySource+1;
	END_IF		

(*******************************************************************************************************************************************)
(* Wort 14*)
(*******************************************************************************************************************************************)
(* Prüfen, ob Wort kopiert werden soll *)
	IF (IN_bCountWords >= 14) THEN
	(* Arraybereich kopieren *)
		OUT_wTargetWord14.0:=IN_pbArraySource^;
		IN_pbArraySource:=IN_pbArraySource+1;
		OUT_wTargetWord14.1:=IN_pbArraySource^;
		IN_pbArraySource:=IN_pbArraySource+1;
		OUT_wTargetWord14.2:=IN_pbArraySource^;
		IN_pbArraySource:=IN_pbArraySource+1;
		OUT_wTargetWord14.3:=IN_pbArraySource^;
		IN_pbArraySource:=IN_pbArraySource+1;
		OUT_wTargetWord14.4:=IN_pbArraySource^;
		IN_pbArraySource:=IN_pbArraySource+1;
		OUT_wTargetWord14.5:=IN_pbArraySource^;
		IN_pbArraySource:=IN_pbArraySource+1;
		OUT_wTargetWord14.6:=IN_pbArraySource^;
		IN_pbArraySource:=IN_pbArraySource+1;
		OUT_wTargetWord14.7:=IN_pbArraySource^;
		IN_pbArraySource:=IN_pbArraySource+1;
		OUT_wTargetWord14.8:=IN_pbArraySource^;
		IN_pbArraySource:=IN_pbArraySource+1;
		OUT_wTargetWord14.9:=IN_pbArraySource^;
		IN_pbArraySource:=IN_pbArraySource+1;
		OUT_wTargetWord14.10:=IN_pbArraySource^;
		IN_pbArraySource:=IN_pbArraySource+1;
		OUT_wTargetWord14.11:=IN_pbArraySource^;
		IN_pbArraySource:=IN_pbArraySource+1;
		OUT_wTargetWord14.12:=IN_pbArraySource^;
		IN_pbArraySource:=IN_pbArraySource+1;
		OUT_wTargetWord14.13:=IN_pbArraySource^;
		IN_pbArraySource:=IN_pbArraySource+1;
		OUT_wTargetWord14.14:=IN_pbArraySource^;
		IN_pbArraySource:=IN_pbArraySource+1;
		OUT_wTargetWord14.15:=IN_pbArraySource^;
		IN_pbArraySource:=IN_pbArraySource+1;
	END_IF	

(*******************************************************************************************************************************************)
(* Wort 15*)
(*******************************************************************************************************************************************)
(* Prüfen, ob Wort kopiert werden soll *)
	IF (IN_bCountWords >= 15) THEN
	(* Arraybereich kopieren *)
		OUT_wTargetWord15.0:=IN_pbArraySource^;
		IN_pbArraySource:=IN_pbArraySource+1;
		OUT_wTargetWord15.1:=IN_pbArraySource^;
		IN_pbArraySource:=IN_pbArraySource+1;
		OUT_wTargetWord15.2:=IN_pbArraySource^;
		IN_pbArraySource:=IN_pbArraySource+1;
		OUT_wTargetWord15.3:=IN_pbArraySource^;
		IN_pbArraySource:=IN_pbArraySource+1;
		OUT_wTargetWord15.4:=IN_pbArraySource^;
		IN_pbArraySource:=IN_pbArraySource+1;
		OUT_wTargetWord15.5:=IN_pbArraySource^;
		IN_pbArraySource:=IN_pbArraySource+1;
		OUT_wTargetWord15.6:=IN_pbArraySource^;
		IN_pbArraySource:=IN_pbArraySource+1;
		OUT_wTargetWord15.7:=IN_pbArraySource^;
		IN_pbArraySource:=IN_pbArraySource+1;
		OUT_wTargetWord15.8:=IN_pbArraySource^;
		IN_pbArraySource:=IN_pbArraySource+1;
		OUT_wTargetWord15.9:=IN_pbArraySource^;
		IN_pbArraySource:=IN_pbArraySource+1;
		OUT_wTargetWord15.10:=IN_pbArraySource^;
		IN_pbArraySource:=IN_pbArraySource+1;
		OUT_wTargetWord15.11:=IN_pbArraySource^;
		IN_pbArraySource:=IN_pbArraySource+1;
		OUT_wTargetWord15.12:=IN_pbArraySource^;
		IN_pbArraySource:=IN_pbArraySource+1;
		OUT_wTargetWord15.13:=IN_pbArraySource^;
		IN_pbArraySource:=IN_pbArraySource+1;
		OUT_wTargetWord15.14:=IN_pbArraySource^;
		IN_pbArraySource:=IN_pbArraySource+1;
		OUT_wTargetWord15.15:=IN_pbArraySource^;
		IN_pbArraySource:=IN_pbArraySource+1;
	END_IF	

(*******************************************************************************************************************************************)
(* Wort 16*)
(*******************************************************************************************************************************************)
(* Prüfen, ob Wort kopiert werden soll *)
	IF (IN_bCountWords >= 16) THEN
	(* Arraybereich kopieren *)
		OUT_wTargetWord16.0:=IN_pbArraySource^;
		IN_pbArraySource:=IN_pbArraySource+1;
		OUT_wTargetWord16.1:=IN_pbArraySource^;
		IN_pbArraySource:=IN_pbArraySource+1;
		OUT_wTargetWord16.2:=IN_pbArraySource^;
		IN_pbArraySource:=IN_pbArraySource+1;
		OUT_wTargetWord16.3:=IN_pbArraySource^;
		IN_pbArraySource:=IN_pbArraySource+1;
		OUT_wTargetWord16.4:=IN_pbArraySource^;
		IN_pbArraySource:=IN_pbArraySource+1;
		OUT_wTargetWord16.5:=IN_pbArraySource^;
		IN_pbArraySource:=IN_pbArraySource+1;
		OUT_wTargetWord16.6:=IN_pbArraySource^;
		IN_pbArraySource:=IN_pbArraySource+1;
		OUT_wTargetWord16.7:=IN_pbArraySource^;
		IN_pbArraySource:=IN_pbArraySource+1;
		OUT_wTargetWord16.8:=IN_pbArraySource^;
		IN_pbArraySource:=IN_pbArraySource+1;
		OUT_wTargetWord16.9:=IN_pbArraySource^;
		IN_pbArraySource:=IN_pbArraySource+1;
		OUT_wTargetWord16.10:=IN_pbArraySource^;
		IN_pbArraySource:=IN_pbArraySource+1;
		OUT_wTargetWord16.11:=IN_pbArraySource^;
		IN_pbArraySource:=IN_pbArraySource+1;
		OUT_wTargetWord16.12:=IN_pbArraySource^;
		IN_pbArraySource:=IN_pbArraySource+1;
		OUT_wTargetWord16.13:=IN_pbArraySource^;
		IN_pbArraySource:=IN_pbArraySource+1;
		OUT_wTargetWord16.14:=IN_pbArraySource^;
		IN_pbArraySource:=IN_pbArraySource+1;
		OUT_wTargetWord16.15:=IN_pbArraySource^;
		IN_pbArraySource:=IN_pbArraySource+1;
END_IF

END_FUNCTION_BLOCK

// ReadMe
PROGRAM ReadMe
VAR
END_VAR

(*
German translation see below

This library project serves as a template for creating your own library that corresponds to the Bosch Rexroth style guide.
This styleguide is stored in the Styleguide folder as a PDF document.
The folder structures corresponding to the style guide already contain objects that can either be adapted to the library function or have to be deleted.
To make the syntax of the reStructuredText easier to understand, some examples have been provided in the declaration part of the MyFB function module, which is located below the MyFunctionality/POUs folder.
Particular attention must be paid to spaces and blank lines in order to ensure the desired formatting results.
For more information, see the web-based online help at https://help.codesys.com/webapp/_cds_guidelines_for_creating_libraries

Recommended procedure for creating a general library:
- Open Library Template
- Save the library template using "File/Save Project As...". Select the name according to the library name.
- Adjustments in the Project Information/Summary object:
   company
   title
   version
   library categories
   author
   Description 
- Adaptation of the "Placeholder" key in the project information/properties object:
  If there is a placeholder in a device description file for this library, it must be entered here as a value. 
  Example: For the library CXA_CommonTypes there is the placeholder CXA_COMMONTYPES, which is resolved in the device description file of ctrlX.
  Thus this placeholder CXA_COMMONTYPES has to be entered as text type in the field "Value" and has to be taken over via the button "Modify". 
  Background: If this library is inserted in the library manager of the general POU, it is automatically inserted as placeholder.

  If there is no placeholder for the library to be created, the "Placeholder" key must be removed from the project information.
  
- Option "Automatically create 'library information' POUs: This option creates functions that allow access to project properties. 
                                                           If these are not required, this option should not be activated.    
- Delete all unneeded objects
- Delete the Styleguide folder
- Delete the ReadMe file
- Customize and save the file History.txt in the _History folder
- After the functionality has been implemented: 
  Execute the command "Build/check all pool objects" and correct any errors.
  If the translation was error and warning free: Execute command "Save project as compiled library...".
- Testing the library: 
  In the test project, install the translated library via the library manager.
  If it was already inserted in the library manager, it is automatically reloaded (only if the library version is the same).
  The non-compiled library can also be installed for debugging purposes.

Dieses Bibliotheksprojekt dient als Vorlage zur Erstellung einer eigenen Bibliothek, die dem Styleguide von Bosch Rexroth entspricht.
Dieser Styleguide liegt im Ordner Styleguide als PDF-Dokument ab.
Die dem Styleguide entsprechenden Ordnerstrukturen enthalten bereits Objekte, die entweder an die eigene Bibliotheksfunktion angepasst werden können oder gelöscht werden müssen.
Um einen einfacheren Einstieg in die Syntax des reStructuredText zu ermöglichen, wurden im Deklarationsteil des Funktionsbausteins MyFB, der sich unterhalb des Ordners MyFunctionality/POUs befindet, einige Beispiele angegeben.
Insbesondere sind auf Leerzeichen und Leerzeilen zu achten, um die gewünschten Formatierungsergebnisse zu gewährleisten.
Weitere Informationen siehe webbasierte Onlinehilfe unter https://help.codesys.com/webapp/_cds_guidelines_for_creating_libraries

Empfohlene Vorgehensweise zur Erstellung einer allgemeinen Bibliothek:
- Bibliotheksvorlage öffnen
- Bibliotheksvorlage mittels "File/Save Project As..." abspeichern. Dabei den Namen entsprechend der Bibliotheksbezeichnung wählen.
- Anpassungen im Objekt Projektinformationen/Zusammenfassung:
  Firma
  Titel
  Version
  Kategorien: Aus bereitgestellter XML-Beschreibungsdatei oder aus einer anderen Library auswählen. Es ist möglich, eigene Kategorien zu erstellen. Siehe Ordner Library category.
  Autor
  Beschreibung 
- Anpassung des Schlüssels "Placeholder" im Objekt Projektinformationen/Eigenschaften: 
  Wenn es ein Platzhalter in einer Gerätebeschreibungsdatei für diese Bibliothek gibt, so ist dieser als Wert hier einzutragen. 
  Beispiel: Für die Bibliothek CXA_CommonTypes gibt es den Platzhalter CXA_COMMONTYPES, der in der Gerätebeschreibungsdatei der ctrlX aufgelöst wird.
  Somit ist dieser Platzhalter CXA_COMMONTYPES als Texttype im Feld "Wert" einzutragen und über den Button "Modify" zu übernehmen. 
  Hintergrund: Wird diese Bibliothek im Bibliotheksverwalter eingefügt, so wird diese bereits als Platzhalterauflösung eingefügt.
  Sollte es für die zu erstellende Bibliothek keinen Platzhalter geben, ist der Schlüssel "Placeholder" aus den Projektinformationen zu entfernen.

- Option "Automatisch 'Bibliotheksinformationen'-POUs erzeugen: Diese Option erzeugt Funktionen, die einen Zugriff auf Projekteigenschaften erlauben. 
                                                                Werden diese nicht benötigt, so sollte diese Option nicht akiviert werden.     
  
- Alle nichtbenötigten Objekte und Ordner löschen
- Den Ordner Styleguide (can be removed) löschen
- Den Ordner Library category (can be removed) löschen
- Diese POU ReadMe löschen
- Das File History.txt im Ordner _History anpassen und speichern
- Nachdem die Funktionalität implementiert worden ist: 
  Kommando "Erstellen/Überprüfe all Poolobjekte" ausführen, ggf. Fehler beheben
  Wenn fehler- und warnungsfrei übersetzt worden ist: Kommando "Datei/Projekt als übersetzte Bibliothek speichern..." ausführen
- Testen der Bibliothek: 
  Im Testprojekt über den Bibliotheksverwalter die übersetzte Bibliothek installieren. 
  Wenn sie bereits im Bibliotheksverwalter eingefügt war, wird sie automatisch neu geladen (nur bei gleicher Bibliotheksversion).
  Für Debugzwecke kann auch die nichtübersetzte Bibliothek installiert werden.

*)

END_PROGRAM

// _History/_History_
(*

Modification - History
""""""""""""""""""""""
========   =========
Version:   0.7.0.0
Name   :   DC-AE/ESW4 (MD)
Date   :   2024-Oct-07
Comment:   - changed categories in LibraryCategory.libcat.xml
-----------------------------------
Version:   0.6.0.0
Name   :   DC-AE/ESW4 (MD)
Date   :   2024-Apr-24
Comment:   - Added Styleguide in english languague
-----------------------------------
Version:   0.5.0.0
Name   :   DC-AE/ESW4 (MD)
Date   :   2023-Nov-07
Comment:   - Bug 749468: ctrlX PLC Engineering: Bibliothekstemplate updaten bzgl. {attribute 'to_string'}
-----------------------------------
Version:   0.4.0.0
Name   :   DC-AE/ESW4 (MD)
Date   :   2023-Nov-03
Comment:   - udpate LibraryCategory.libcat.xml
-----------------------------------
Version:   0.3.0.0
Name   :   DC-AE/ESW4 (MD)
Date   :   2023-Feb-15
Comment:   - added _History_ as a program
           - udpate Styleguide
           - removed/added some properties of projectinformation
-----------------------------------
Version:   0.2.0.0
Name   :   DC-AE/ESW4 (MD)
Date   :   2022-Oct-21
Comment:   - added Folder Library category
           - removed category in project information
-----------------------------------
Version:   0.1.0.0
Name   :   DC-AE/ESW4 (4+4)
Date   :   2020-Nov-11
Comment:   -Bug 240837:
	   - added CXA_Utilities and CXA_CommonTypes to library manager
           - update of Styleguide.pdf
           - library compatibility changed to ctrlX PLC 1.5.1
-----------------------------------
Version:   0.1.0.0
Name   :   DC-AE/ESW4 (4+4)
Date   :   2019-Sep-26
Comment:   - 1st version 

========   =========

*)
PROGRAM _History_
VAR
END_VAR

END_PROGRAM

// _Library Informations/GetLibVersion
// This function has been automatically generated from the project information.
FUNCTION GetLibVersion : VERSION
VAR_INPUT
	
END_VAR

GetLibVersion.uiMajor := 0;
GetLibVersion.uiMinor := 7;
GetLibVersion.uiServicePack := 0;
GetLibVersion.uiPatch := 1;

END_FUNCTION

// _Library Informations/GetLibVersionNumber
// This function has been automatically generated from the project information.
FUNCTION GetLibVersionNumber : DWORD
VAR_INPUT
	
END_VAR

GetLibVersionNumber := 458753;

END_FUNCTION

// GeneralFunctionBlocks/FB_ArrayToWord
{attribute 'qualified_only'}
{attribute 'namespace' := 'ILGStdLib.FunctionBlocks.' }
FUNCTION_BLOCK FB_ArrayToWord
(*####################################################################################################################################################
	
	Kurzbeschreibung:
		Funktionsbaustein zum Kopieren eines Arraybereichs in Variablen vom Datentyp WORD.

	Beschreibung:
		Am Eingang "iArray_Quelle_i" wird das zu kopierende Array parametriert. Über den Eingang "iStart_Offset_i" kann ein Offset 
		bezogen auf das am Eingang "iArray_Quelle_i" angegebene Array angegeben werden. Wird als "iStart_Offset_i" "0" angegeben so startet der 
		Kopiervorgang am ersten Feld des Eingang "iArray_Quelle_i".
		Der Eingang "iAnzahl_Worte_i" gibt die Anzahl der zu kopierende Worte bezogen auf den "iStart_Offset_i" an.
		An den Ausgängen "wZiel_Wort_1_o" ...."wZiel_Wort_16_o" können die Arrayinformationen Wortweise abgegriffen werden.
		
*******************************************************************************************************************************************************
	Historie:
		---------------------------------------------------------------------------------------------------------------------------------------------
		|	Datum			|		Name			|	Beschreibung																				|
		---------------------------------------------------------------------------------------------------------------------------------------------																						
		|	30.5.2011		|		T.Hauser		|	Baustein neu erstellt																		|
		---------------------------------------------------------------------------------------------------------------------------------------------
		|					|						|																								|
		---------------------------------------------------------------------------------------------------------------------------------------------
		|					|						|																								|
		---------------------------------------------------------------------------------------------------------------------------------------------
		|					|						|																								|
		---------------------------------------------------------------------------------------------------------------------------------------------

########################################################################################################################################################*)



(*******************************************************************************************************************************************)
(* Eingangsvariablen *)
(*******************************************************************************************************************************************)		
VAR_INPUT
	IN_pbArraySource:			POINTER TO BOOL;	(* Array aus dem der Datenbereich kopiert werden soll. Angabe ohne Index *)
	IN_bStartOffset:			BYTE; 				(* Defnition des ersten zu kopierenden Wert vom Eingang "iArray_Quelle_i" *)
	IN_bCountWords:				BYTE; 				(* Anzahl Worte die kopiert werden sollen*)
END_VAR

(*******************************************************************************************************************************************)
(* Ausgangsvariablen *)
(*******************************************************************************************************************************************)
VAR_OUTPUT
	OUT_wTargetWord1:				WORD;				(*Ziel Wort Bereich 1*)
	OUT_wTargetWord2:				WORD;				(*Ziel Wort Bereich 2*)
	OUT_wTargetWord3:				WORD;				(*Ziel Wort Bereich 3*)	
	OUT_wTargetWord4:				WORD;				(*Ziel Wort Bereich 4*)
	OUT_wTargetWord5:				WORD;				(*Ziel Wort Bereich 5*)
	OUT_wTargetWord6:				WORD;				(*Ziel Wort Bereich 6*)	
	OUT_wTargetWord7:				WORD;				(*Ziel Wort Bereich 7*)
	OUT_wTargetWord8:				WORD;				(*Ziel Wort Bereich 8*)
	OUT_wTargetWord9:				WORD;				(*Ziel Wort Bereich 9*)	
	OUT_wTargetWord10:				WORD;				(*Ziel Wort Bereich 10*)
	OUT_wTargetWord11:				WORD;				(*Ziel Wort Bereich 11*)
	OUT_wTargetWord12:				WORD;				(*Ziel Wort Bereich 12*)
	OUT_wTargetWord13:				WORD;				(*Ziel Wort Bereich 13*)	
	OUT_wTargetWord14:				WORD;				(*Ziel Wort Bereich 14*)
	OUT_wTargetWord15:				WORD;				(*Ziel Wort Bereich 15*)
	OUT_wTargetWord16:				WORD;				(*Ziel Wort Bereich 16*)
END_VAR

(*******************************************************************************************************************************************)
(* Interne Variablen *)
(*******************************************************************************************************************************************)
VAR
END_VAR

(* Anzahl der zu kopierenden Worte begrenzen *)
	IF IN_bCountWords > 16 THEN
		IN_bCountWords:= 16;
	END_IF

(* Startadresse vorbelegen*)
	IN_pbArraySource:= IN_pbArraySource + IN_bStartOffset;
(*******************************************************************************************************************************************)
(* Wort 1*)
(*******************************************************************************************************************************************)
(* Prüfen, ob Wort kopiert werden soll *)
	IF (IN_bCountWords >= 1) THEN
		(* Arraybereich kopieren *)
			OUT_wTargetWord1.0:=IN_pbArraySource^;
			IN_pbArraySource:=IN_pbArraySource+1;
			OUT_wTargetWord1.1:=IN_pbArraySource^;
			IN_pbArraySource:=IN_pbArraySource+1;
			OUT_wTargetWord1.2:=IN_pbArraySource^;
			IN_pbArraySource:=IN_pbArraySource+1;
			OUT_wTargetWord1.3:=IN_pbArraySource^;
			IN_pbArraySource:=IN_pbArraySource+1;
			OUT_wTargetWord1.4:=IN_pbArraySource^;
			IN_pbArraySource:=IN_pbArraySource+1;
			OUT_wTargetWord1.5:=IN_pbArraySource^;
			IN_pbArraySource:=IN_pbArraySource+1;
			OUT_wTargetWord1.6:=IN_pbArraySource^;
			IN_pbArraySource:=IN_pbArraySource+1;
			OUT_wTargetWord1.7:=IN_pbArraySource^;
			IN_pbArraySource:=IN_pbArraySource+1;
			OUT_wTargetWord1.8:=IN_pbArraySource^;
			IN_pbArraySource:=IN_pbArraySource+1;
			OUT_wTargetWord1.9:=IN_pbArraySource^;
			IN_pbArraySource:=IN_pbArraySource+1;
			OUT_wTargetWord1.10:=IN_pbArraySource^;
			IN_pbArraySource:=IN_pbArraySource+1;
			OUT_wTargetWord1.11:=IN_pbArraySource^;
			IN_pbArraySource:=IN_pbArraySource+1;
			OUT_wTargetWord1.12:=IN_pbArraySource^;
			IN_pbArraySource:=IN_pbArraySource+1;
			OUT_wTargetWord1.13:=IN_pbArraySource^;
			IN_pbArraySource:=IN_pbArraySource+1;
			OUT_wTargetWord1.14:=IN_pbArraySource^;
			IN_pbArraySource:=IN_pbArraySource+1;
			OUT_wTargetWord1.15:=IN_pbArraySource^;
			IN_pbArraySource:=IN_pbArraySource+1;
	END_IF

(*******************************************************************************************************************************************)
(* Wort 2*)
(*******************************************************************************************************************************************)
(* Prüfen, ob Wort kopiert werden soll *)
	IF (IN_bCountWords >= 2) THEN
		(* Arraybereich kopieren *)
			OUT_wTargetWord2.0:=IN_pbArraySource^;
			IN_pbArraySource:=IN_pbArraySource+1;
			OUT_wTargetWord2.1:=IN_pbArraySource^;
			IN_pbArraySource:=IN_pbArraySource+1;
			OUT_wTargetWord2.2:=IN_pbArraySource^;
			IN_pbArraySource:=IN_pbArraySource+1;
			OUT_wTargetWord2.3:=IN_pbArraySource^;
			IN_pbArraySource:=IN_pbArraySource+1;
			OUT_wTargetWord2.4:=IN_pbArraySource^;
			IN_pbArraySource:=IN_pbArraySource+1;
			OUT_wTargetWord2.5:=IN_pbArraySource^;
			IN_pbArraySource:=IN_pbArraySource+1;
			OUT_wTargetWord2.6:=IN_pbArraySource^;
			IN_pbArraySource:=IN_pbArraySource+1;
			OUT_wTargetWord2.7:=IN_pbArraySource^;
			IN_pbArraySource:=IN_pbArraySource+1;
			OUT_wTargetWord2.8:=IN_pbArraySource^;
			IN_pbArraySource:=IN_pbArraySource+1;
			OUT_wTargetWord2.9:=IN_pbArraySource^;
			IN_pbArraySource:=IN_pbArraySource+1;
			OUT_wTargetWord2.10:=IN_pbArraySource^;
			IN_pbArraySource:=IN_pbArraySource+1;
			OUT_wTargetWord2.11:=IN_pbArraySource^;
			IN_pbArraySource:=IN_pbArraySource+1;
			OUT_wTargetWord2.12:=IN_pbArraySource^;
			IN_pbArraySource:=IN_pbArraySource+1;
			OUT_wTargetWord2.13:=IN_pbArraySource^;
			IN_pbArraySource:=IN_pbArraySource+1;
			OUT_wTargetWord2.14:=IN_pbArraySource^;
			IN_pbArraySource:=IN_pbArraySource+1;
			OUT_wTargetWord2.15:=IN_pbArraySource^;
			IN_pbArraySource:=IN_pbArraySource+1;
	END_IF		
		
(*******************************************************************************************************************************************)
(* Wort 3*)
(*******************************************************************************************************************************************)
(* Prüfen, ob Wort kopiert werden soll *)
	IF (IN_bCountWords >= 3) THEN
	(* Arraybereich kopieren *)
		OUT_wTargetWord3.0:=IN_pbArraySource^;
		IN_pbArraySource:=IN_pbArraySource+1;
		OUT_wTargetWord3.1:=IN_pbArraySource^;
		IN_pbArraySource:=IN_pbArraySource+1;
		OUT_wTargetWord3.2:=IN_pbArraySource^;
		IN_pbArraySource:=IN_pbArraySource+1;
		OUT_wTargetWord3.3:=IN_pbArraySource^;
		IN_pbArraySource:=IN_pbArraySource+1;
		OUT_wTargetWord3.4:=IN_pbArraySource^;
		IN_pbArraySource:=IN_pbArraySource+1;
		OUT_wTargetWord3.5:=IN_pbArraySource^;
		IN_pbArraySource:=IN_pbArraySource+1;
		OUT_wTargetWord3.6:=IN_pbArraySource^;
		IN_pbArraySource:=IN_pbArraySource+1;
		OUT_wTargetWord3.7:=IN_pbArraySource^;
		IN_pbArraySource:=IN_pbArraySource+1;
		OUT_wTargetWord3.8:=IN_pbArraySource^;
		IN_pbArraySource:=IN_pbArraySource+1;
		OUT_wTargetWord3.9:=IN_pbArraySource^;
		IN_pbArraySource:=IN_pbArraySource+1;
		OUT_wTargetWord3.10:=IN_pbArraySource^;
		IN_pbArraySource:=IN_pbArraySource+1;
		OUT_wTargetWord3.11:=IN_pbArraySource^;
		IN_pbArraySource:=IN_pbArraySource+1;
		OUT_wTargetWord3.12:=IN_pbArraySource^;
		IN_pbArraySource:=IN_pbArraySource+1;
		OUT_wTargetWord3.13:=IN_pbArraySource^;
		IN_pbArraySource:=IN_pbArraySource+1;
		OUT_wTargetWord3.14:=IN_pbArraySource^;
		IN_pbArraySource:=IN_pbArraySource+1;
		OUT_wTargetWord3.15:=IN_pbArraySource^;
		IN_pbArraySource:=IN_pbArraySource+1;
	END_IF		
	
(*******************************************************************************************************************************************)
(* Wort 4*)
(*******************************************************************************************************************************************)
(* Prüfen, ob Wort kopiert werden soll *)
	IF (IN_bCountWords >= 4) THEN
	(* Arraybereich kopieren *)
		OUT_wTargetWord4.0:=IN_pbArraySource^;
		IN_pbArraySource:=IN_pbArraySource+1;
		OUT_wTargetWord4.1:=IN_pbArraySource^;
		IN_pbArraySource:=IN_pbArraySource+1;
		OUT_wTargetWord4.2:=IN_pbArraySource^;
		IN_pbArraySource:=IN_pbArraySource+1;
		OUT_wTargetWord4.3:=IN_pbArraySource^;
		IN_pbArraySource:=IN_pbArraySource+1;
		OUT_wTargetWord4.4:=IN_pbArraySource^;
		IN_pbArraySource:=IN_pbArraySource+1;
		OUT_wTargetWord4.5:=IN_pbArraySource^;
		IN_pbArraySource:=IN_pbArraySource+1;
		OUT_wTargetWord4.6:=IN_pbArraySource^;
		IN_pbArraySource:=IN_pbArraySource+1;
		OUT_wTargetWord4.7:=IN_pbArraySource^;
		IN_pbArraySource:=IN_pbArraySource+1;
		OUT_wTargetWord4.8:=IN_pbArraySource^;
		IN_pbArraySource:=IN_pbArraySource+1;
		OUT_wTargetWord4.9:=IN_pbArraySource^;
		IN_pbArraySource:=IN_pbArraySource+1;
		OUT_wTargetWord4.10:=IN_pbArraySource^;
		IN_pbArraySource:=IN_pbArraySource+1;
		OUT_wTargetWord4.11:=IN_pbArraySource^;
		IN_pbArraySource:=IN_pbArraySource+1;
		OUT_wTargetWord4.12:=IN_pbArraySource^;
		IN_pbArraySource:=IN_pbArraySource+1;
		OUT_wTargetWord4.13:=IN_pbArraySource^;
		IN_pbArraySource:=IN_pbArraySource+1;
		OUT_wTargetWord4.14:=IN_pbArraySource^;
		IN_pbArraySource:=IN_pbArraySource+1;
		OUT_wTargetWord4.15:=IN_pbArraySource^;
		IN_pbArraySource:=IN_pbArraySource+1;
	END_IF			

(*******************************************************************************************************************************************)
(* Wort 5*)
(*******************************************************************************************************************************************)
(* Prüfen, ob Wort kopiert werden soll *)
	IF (IN_bCountWords >= 5) THEN
	(* Arraybereich kopieren *)
		OUT_wTargetWord5.0:=IN_pbArraySource^;
		IN_pbArraySource:=IN_pbArraySource+1;
		OUT_wTargetWord5.1:=IN_pbArraySource^;
		IN_pbArraySource:=IN_pbArraySource+1;
		OUT_wTargetWord5.2:=IN_pbArraySource^;
		IN_pbArraySource:=IN_pbArraySource+1;
		OUT_wTargetWord5.3:=IN_pbArraySource^;
		IN_pbArraySource:=IN_pbArraySource+1;
		OUT_wTargetWord5.4:=IN_pbArraySource^;
		IN_pbArraySource:=IN_pbArraySource+1;
		OUT_wTargetWord5.5:=IN_pbArraySource^;
		IN_pbArraySource:=IN_pbArraySource+1;
		OUT_wTargetWord5.6:=IN_pbArraySource^;
		IN_pbArraySource:=IN_pbArraySource+1;
		OUT_wTargetWord5.7:=IN_pbArraySource^;
		IN_pbArraySource:=IN_pbArraySource+1;
		OUT_wTargetWord5.8:=IN_pbArraySource^;
		IN_pbArraySource:=IN_pbArraySource+1;
		OUT_wTargetWord5.9:=IN_pbArraySource^;
		IN_pbArraySource:=IN_pbArraySource+1;
		OUT_wTargetWord5.10:=IN_pbArraySource^;
		IN_pbArraySource:=IN_pbArraySource+1;
		OUT_wTargetWord5.11:=IN_pbArraySource^;
		IN_pbArraySource:=IN_pbArraySource+1;
		OUT_wTargetWord5.12:=IN_pbArraySource^;
		IN_pbArraySource:=IN_pbArraySource+1;
		OUT_wTargetWord5.13:=IN_pbArraySource^;
		IN_pbArraySource:=IN_pbArraySource+1;
		OUT_wTargetWord5.14:=IN_pbArraySource^;
		IN_pbArraySource:=IN_pbArraySource+1;
		OUT_wTargetWord5.15:=IN_pbArraySource^;
		IN_pbArraySource:=IN_pbArraySource+1;
	END_IF			

(*******************************************************************************************************************************************)
(* Wort 6*)
(*******************************************************************************************************************************************)
(* Prüfen, ob Wort kopiert werden soll *)
	IF (IN_bCountWords >= 6) THEN
	(* Arraybereich kopieren *)
		OUT_wTargetWord6.0:=IN_pbArraySource^;
		IN_pbArraySource:=IN_pbArraySource+1;
		OUT_wTargetWord6.1:=IN_pbArraySource^;
		IN_pbArraySource:=IN_pbArraySource+1;
		OUT_wTargetWord6.2:=IN_pbArraySource^;
		IN_pbArraySource:=IN_pbArraySource+1;
		OUT_wTargetWord6.3:=IN_pbArraySource^;
		IN_pbArraySource:=IN_pbArraySource+1;
		OUT_wTargetWord6.4:=IN_pbArraySource^;
		IN_pbArraySource:=IN_pbArraySource+1;
		OUT_wTargetWord6.5:=IN_pbArraySource^;
		IN_pbArraySource:=IN_pbArraySource+1;
		OUT_wTargetWord6.6:=IN_pbArraySource^;
		IN_pbArraySource:=IN_pbArraySource+1;
		OUT_wTargetWord6.7:=IN_pbArraySource^;
		IN_pbArraySource:=IN_pbArraySource+1;
		OUT_wTargetWord6.8:=IN_pbArraySource^;
		IN_pbArraySource:=IN_pbArraySource+1;
		OUT_wTargetWord6.9:=IN_pbArraySource^;
		IN_pbArraySource:=IN_pbArraySource+1;
		OUT_wTargetWord6.10:=IN_pbArraySource^;
		IN_pbArraySource:=IN_pbArraySource+1;
		OUT_wTargetWord6.11:=IN_pbArraySource^;
		IN_pbArraySource:=IN_pbArraySource+1;
		OUT_wTargetWord6.12:=IN_pbArraySource^;
		IN_pbArraySource:=IN_pbArraySource+1;
		OUT_wTargetWord6.13:=IN_pbArraySource^;
		IN_pbArraySource:=IN_pbArraySource+1;
		OUT_wTargetWord6.14:=IN_pbArraySource^;
		IN_pbArraySource:=IN_pbArraySource+1;
		OUT_wTargetWord6.15:=IN_pbArraySource^;
		IN_pbArraySource:=IN_pbArraySource+1;
END_IF
		
(*******************************************************************************************************************************************)
(* Wort 7*)
(*******************************************************************************************************************************************)
(* Prüfen, ob Wort kopiert werden soll *)
	IF (IN_bCountWords >= 7) THEN
	(* Arraybereich kopieren *)
		OUT_wTargetWord7.0:=IN_pbArraySource^;
		IN_pbArraySource:=IN_pbArraySource+1;
		OUT_wTargetWord7.1:=IN_pbArraySource^;
		IN_pbArraySource:=IN_pbArraySource+1;
		OUT_wTargetWord7.2:=IN_pbArraySource^;
		IN_pbArraySource:=IN_pbArraySource+1;
		OUT_wTargetWord7.3:=IN_pbArraySource^;
		IN_pbArraySource:=IN_pbArraySource+1;
		OUT_wTargetWord7.4:=IN_pbArraySource^;
		IN_pbArraySource:=IN_pbArraySource+1;
		OUT_wTargetWord7.5:=IN_pbArraySource^;
		IN_pbArraySource:=IN_pbArraySource+1;
		OUT_wTargetWord7.6:=IN_pbArraySource^;
		IN_pbArraySource:=IN_pbArraySource+1;
		OUT_wTargetWord7.7:=IN_pbArraySource^;
		IN_pbArraySource:=IN_pbArraySource+1;
		OUT_wTargetWord7.8:=IN_pbArraySource^;
		IN_pbArraySource:=IN_pbArraySource+1;
		OUT_wTargetWord7.9:=IN_pbArraySource^;
		IN_pbArraySource:=IN_pbArraySource+1;
		OUT_wTargetWord7.10:=IN_pbArraySource^;
		IN_pbArraySource:=IN_pbArraySource+1;
		OUT_wTargetWord7.11:=IN_pbArraySource^;
		IN_pbArraySource:=IN_pbArraySource+1;
		OUT_wTargetWord7.12:=IN_pbArraySource^;
		IN_pbArraySource:=IN_pbArraySource+1;
		OUT_wTargetWord7.13:=IN_pbArraySource^;
		IN_pbArraySource:=IN_pbArraySource+1;
		OUT_wTargetWord7.14:=IN_pbArraySource^;
		IN_pbArraySource:=IN_pbArraySource+1;
		OUT_wTargetWord7.15:=IN_pbArraySource^;
		IN_pbArraySource:=IN_pbArraySource+1;
	END_IF	
		
(*******************************************************************************************************************************************)
(* Wort 8*)
(*******************************************************************************************************************************************)
(* Prüfen, ob Wort kopiert werden soll *)
	IF (IN_bCountWords >= 8) THEN
	(* Arraybereich kopieren *)
		OUT_wTargetWord8.0:=IN_pbArraySource^;
		IN_pbArraySource:=IN_pbArraySource+1;
		OUT_wTargetWord8.1:=IN_pbArraySource^;
		IN_pbArraySource:=IN_pbArraySource+1;
		OUT_wTargetWord8.2:=IN_pbArraySource^;
		IN_pbArraySource:=IN_pbArraySource+1;
		OUT_wTargetWord8.3:=IN_pbArraySource^;
		IN_pbArraySource:=IN_pbArraySource+1;
		OUT_wTargetWord8.4:=IN_pbArraySource^;
		IN_pbArraySource:=IN_pbArraySource+1;
		OUT_wTargetWord8.5:=IN_pbArraySource^;
		IN_pbArraySource:=IN_pbArraySource+1;
		OUT_wTargetWord8.6:=IN_pbArraySource^;
		IN_pbArraySource:=IN_pbArraySource+1;
		OUT_wTargetWord8.7:=IN_pbArraySource^;
		IN_pbArraySource:=IN_pbArraySource+1;
		OUT_wTargetWord8.8:=IN_pbArraySource^;
		IN_pbArraySource:=IN_pbArraySource+1;
		OUT_wTargetWord8.9:=IN_pbArraySource^;
		IN_pbArraySource:=IN_pbArraySource+1;
		OUT_wTargetWord8.10:=IN_pbArraySource^;
		IN_pbArraySource:=IN_pbArraySource+1;
		OUT_wTargetWord8.11:=IN_pbArraySource^;
		IN_pbArraySource:=IN_pbArraySource+1;
		OUT_wTargetWord8.12:=IN_pbArraySource^;
		IN_pbArraySource:=IN_pbArraySource+1;
		OUT_wTargetWord8.13:=IN_pbArraySource^;
		IN_pbArraySource:=IN_pbArraySource+1;
		OUT_wTargetWord8.14:=IN_pbArraySource^;
		IN_pbArraySource:=IN_pbArraySource+1;
		OUT_wTargetWord8.15:=IN_pbArraySource^;
		IN_pbArraySource:=IN_pbArraySource+1;
	END_IF	

(*******************************************************************************************************************************************)
(* Wort 9*)
(*******************************************************************************************************************************************)
(* Prüfen, ob Wort kopiert werden soll *)
	IF (IN_bCountWords >= 9) THEN
	(* Arraybereich kopieren *)
		OUT_wTargetWord9.0:=IN_pbArraySource^;
		IN_pbArraySource:=IN_pbArraySource+1;
		OUT_wTargetWord9.1:=IN_pbArraySource^;
		IN_pbArraySource:=IN_pbArraySource+1;
		OUT_wTargetWord9.2:=IN_pbArraySource^;
		IN_pbArraySource:=IN_pbArraySource+1;
		OUT_wTargetWord9.3:=IN_pbArraySource^;
		IN_pbArraySource:=IN_pbArraySource+1;
		OUT_wTargetWord9.4:=IN_pbArraySource^;
		IN_pbArraySource:=IN_pbArraySource+1;
		OUT_wTargetWord9.5:=IN_pbArraySource^;
		IN_pbArraySource:=IN_pbArraySource+1;
		OUT_wTargetWord9.6:=IN_pbArraySource^;
		IN_pbArraySource:=IN_pbArraySource+1;
		OUT_wTargetWord9.7:=IN_pbArraySource^;
		IN_pbArraySource:=IN_pbArraySource+1;
		OUT_wTargetWord9.8:=IN_pbArraySource^;
		IN_pbArraySource:=IN_pbArraySource+1;
		OUT_wTargetWord9.9:=IN_pbArraySource^;
		IN_pbArraySource:=IN_pbArraySource+1;
		OUT_wTargetWord9.10:=IN_pbArraySource^;
		IN_pbArraySource:=IN_pbArraySource+1;
		OUT_wTargetWord9.11:=IN_pbArraySource^;
		IN_pbArraySource:=IN_pbArraySource+1;
		OUT_wTargetWord9.12:=IN_pbArraySource^;
		IN_pbArraySource:=IN_pbArraySource+1;
		OUT_wTargetWord9.13:=IN_pbArraySource^;
		IN_pbArraySource:=IN_pbArraySource+1;
		OUT_wTargetWord9.14:=IN_pbArraySource^;
		IN_pbArraySource:=IN_pbArraySource+1;
		OUT_wTargetWord9.15:=IN_pbArraySource^;
		IN_pbArraySource:=IN_pbArraySource+1;
	END_IF	

(*******************************************************************************************************************************************)
(* Wort 10*)
(*******************************************************************************************************************************************)
(* Prüfen, ob Wort kopiert werden soll *)
	IF (IN_bCountWords >= 10) THEN
	(* Arraybereich kopieren *)
		OUT_wTargetWord10.0:=IN_pbArraySource^;
		IN_pbArraySource:=IN_pbArraySource+1;
		OUT_wTargetWord10.1:=IN_pbArraySource^;
		IN_pbArraySource:=IN_pbArraySource+1;
		OUT_wTargetWord10.2:=IN_pbArraySource^;
		IN_pbArraySource:=IN_pbArraySource+1;
		OUT_wTargetWord10.3:=IN_pbArraySource^;
		IN_pbArraySource:=IN_pbArraySource+1;
		OUT_wTargetWord10.4:=IN_pbArraySource^;
		IN_pbArraySource:=IN_pbArraySource+1;
		OUT_wTargetWord10.5:=IN_pbArraySource^;
		IN_pbArraySource:=IN_pbArraySource+1;
		OUT_wTargetWord10.6:=IN_pbArraySource^;
		IN_pbArraySource:=IN_pbArraySource+1;
		OUT_wTargetWord10.7:=IN_pbArraySource^;
		IN_pbArraySource:=IN_pbArraySource+1;
		OUT_wTargetWord10.8:=IN_pbArraySource^;
		IN_pbArraySource:=IN_pbArraySource+1;
		OUT_wTargetWord10.9:=IN_pbArraySource^;
		IN_pbArraySource:=IN_pbArraySource+1;
		OUT_wTargetWord10.10:=IN_pbArraySource^;
		IN_pbArraySource:=IN_pbArraySource+1;
		OUT_wTargetWord10.11:=IN_pbArraySource^;
		IN_pbArraySource:=IN_pbArraySource+1;
		OUT_wTargetWord10.12:=IN_pbArraySource^;
		IN_pbArraySource:=IN_pbArraySource+1;
		OUT_wTargetWord10.13:=IN_pbArraySource^;
		IN_pbArraySource:=IN_pbArraySource+1;
		OUT_wTargetWord10.14:=IN_pbArraySource^;
		IN_pbArraySource:=IN_pbArraySource+1;
		OUT_wTargetWord10.15:=IN_pbArraySource^;
		IN_pbArraySource:=IN_pbArraySource+1;
	END_IF		

(*******************************************************************************************************************************************)
(* Wort 11*)
(*******************************************************************************************************************************************)
(* Prüfen, ob Wort kopiert werden soll *)
	IF (IN_bCountWords >= 11) THEN
	(* Arraybereich kopieren *)
		OUT_wTargetWord11.0:=IN_pbArraySource^;
		IN_pbArraySource:=IN_pbArraySource+1;
		OUT_wTargetWord11.1:=IN_pbArraySource^;
		IN_pbArraySource:=IN_pbArraySource+1;
		OUT_wTargetWord11.2:=IN_pbArraySource^;
		IN_pbArraySource:=IN_pbArraySource+1;
		OUT_wTargetWord11.3:=IN_pbArraySource^;
		IN_pbArraySource:=IN_pbArraySource+1;
		OUT_wTargetWord11.4:=IN_pbArraySource^;
		IN_pbArraySource:=IN_pbArraySource+1;
		OUT_wTargetWord11.5:=IN_pbArraySource^;
		IN_pbArraySource:=IN_pbArraySource+1;
		OUT_wTargetWord11.6:=IN_pbArraySource^;
		IN_pbArraySource:=IN_pbArraySource+1;
		OUT_wTargetWord11.7:=IN_pbArraySource^;
		IN_pbArraySource:=IN_pbArraySource+1;
		OUT_wTargetWord11.8:=IN_pbArraySource^;
		IN_pbArraySource:=IN_pbArraySource+1;
		OUT_wTargetWord11.9:=IN_pbArraySource^;
		IN_pbArraySource:=IN_pbArraySource+1;
		OUT_wTargetWord11.10:=IN_pbArraySource^;
		IN_pbArraySource:=IN_pbArraySource+1;
		OUT_wTargetWord11.11:=IN_pbArraySource^;
		IN_pbArraySource:=IN_pbArraySource+1;
		OUT_wTargetWord11.12:=IN_pbArraySource^;
		IN_pbArraySource:=IN_pbArraySource+1;
		OUT_wTargetWord11.13:=IN_pbArraySource^;
		IN_pbArraySource:=IN_pbArraySource+1;
		OUT_wTargetWord11.14:=IN_pbArraySource^;
		IN_pbArraySource:=IN_pbArraySource+1;
		OUT_wTargetWord11.15:=IN_pbArraySource^;
		IN_pbArraySource:=IN_pbArraySource+1;
	END_IF		
	
(*******************************************************************************************************************************************)
(* Wort 12*)
(*******************************************************************************************************************************************)
(* Prüfen, ob Wort kopiert werden soll *)
	IF (IN_bCountWords >= 12) THEN
	(* Arraybereich kopieren *)
		OUT_wTargetWord12.0:=IN_pbArraySource^;
		IN_pbArraySource:=IN_pbArraySource+1;
		OUT_wTargetWord12.1:=IN_pbArraySource^;
		IN_pbArraySource:=IN_pbArraySource+1;
		OUT_wTargetWord12.2:=IN_pbArraySource^;
		IN_pbArraySource:=IN_pbArraySource+1;
		OUT_wTargetWord12.3:=IN_pbArraySource^;
		IN_pbArraySource:=IN_pbArraySource+1;
		OUT_wTargetWord12.4:=IN_pbArraySource^;
		IN_pbArraySource:=IN_pbArraySource+1;
		OUT_wTargetWord12.5:=IN_pbArraySource^;
		IN_pbArraySource:=IN_pbArraySource+1;
		OUT_wTargetWord12.6:=IN_pbArraySource^;
		IN_pbArraySource:=IN_pbArraySource+1;
		OUT_wTargetWord12.7:=IN_pbArraySource^;
		IN_pbArraySource:=IN_pbArraySource+1;
		OUT_wTargetWord12.8:=IN_pbArraySource^;
		IN_pbArraySource:=IN_pbArraySource+1;
		OUT_wTargetWord12.9:=IN_pbArraySource^;
		IN_pbArraySource:=IN_pbArraySource+1;
		OUT_wTargetWord12.10:=IN_pbArraySource^;
		IN_pbArraySource:=IN_pbArraySource+1;
		OUT_wTargetWord12.11:=IN_pbArraySource^;
		IN_pbArraySource:=IN_pbArraySource+1;
		OUT_wTargetWord12.12:=IN_pbArraySource^;
		IN_pbArraySource:=IN_pbArraySource+1;
		OUT_wTargetWord12.13:=IN_pbArraySource^;
		IN_pbArraySource:=IN_pbArraySource+1;
		OUT_wTargetWord12.14:=IN_pbArraySource^;
		IN_pbArraySource:=IN_pbArraySource+1;
		OUT_wTargetWord12.15:=IN_pbArraySource^;
		IN_pbArraySource:=IN_pbArraySource+1;
	END_IF	

(*******************************************************************************************************************************************)
(* Wort 13*)
(*******************************************************************************************************************************************)
(* Prüfen, ob Wort kopiert werden soll *)
	IF (IN_bCountWords >= 13) THEN
	(* Arraybereich kopieren *)
		OUT_wTargetWord13.0:=IN_pbArraySource^;
		IN_pbArraySource:=IN_pbArraySource+1;
		OUT_wTargetWord13.1:=IN_pbArraySource^;
		IN_pbArraySource:=IN_pbArraySource+1;
		OUT_wTargetWord13.2:=IN_pbArraySource^;
		IN_pbArraySource:=IN_pbArraySource+1;
		OUT_wTargetWord13.3:=IN_pbArraySource^;
		IN_pbArraySource:=IN_pbArraySource+1;
		OUT_wTargetWord13.4:=IN_pbArraySource^;
		IN_pbArraySource:=IN_pbArraySource+1;
		OUT_wTargetWord13.5:=IN_pbArraySource^;
		IN_pbArraySource:=IN_pbArraySource+1;
		OUT_wTargetWord13.6:=IN_pbArraySource^;
		IN_pbArraySource:=IN_pbArraySource+1;
		OUT_wTargetWord13.7:=IN_pbArraySource^;
		IN_pbArraySource:=IN_pbArraySource+1;
		OUT_wTargetWord13.8:=IN_pbArraySource^;
		IN_pbArraySource:=IN_pbArraySource+1;
		OUT_wTargetWord13.9:=IN_pbArraySource^;
		IN_pbArraySource:=IN_pbArraySource+1;
		OUT_wTargetWord13.10:=IN_pbArraySource^;
		IN_pbArraySource:=IN_pbArraySource+1;
		OUT_wTargetWord13.11:=IN_pbArraySource^;
		IN_pbArraySource:=IN_pbArraySource+1;
		OUT_wTargetWord13.12:=IN_pbArraySource^;
		IN_pbArraySource:=IN_pbArraySource+1;
		OUT_wTargetWord13.13:=IN_pbArraySource^;
		IN_pbArraySource:=IN_pbArraySource+1;
		OUT_wTargetWord13.14:=IN_pbArraySource^;
		IN_pbArraySource:=IN_pbArraySource+1;
		OUT_wTargetWord13.15:=IN_pbArraySource^;
		IN_pbArraySource:=IN_pbArraySource+1;
	END_IF		

(*******************************************************************************************************************************************)
(* Wort 14*)
(*******************************************************************************************************************************************)
(* Prüfen, ob Wort kopiert werden soll *)
	IF (IN_bCountWords >= 14) THEN
	(* Arraybereich kopieren *)
		OUT_wTargetWord14.0:=IN_pbArraySource^;
		IN_pbArraySource:=IN_pbArraySource+1;
		OUT_wTargetWord14.1:=IN_pbArraySource^;
		IN_pbArraySource:=IN_pbArraySource+1;
		OUT_wTargetWord14.2:=IN_pbArraySource^;
		IN_pbArraySource:=IN_pbArraySource+1;
		OUT_wTargetWord14.3:=IN_pbArraySource^;
		IN_pbArraySource:=IN_pbArraySource+1;
		OUT_wTargetWord14.4:=IN_pbArraySource^;
		IN_pbArraySource:=IN_pbArraySource+1;
		OUT_wTargetWord14.5:=IN_pbArraySource^;
		IN_pbArraySource:=IN_pbArraySource+1;
		OUT_wTargetWord14.6:=IN_pbArraySource^;
		IN_pbArraySource:=IN_pbArraySource+1;
		OUT_wTargetWord14.7:=IN_pbArraySource^;
		IN_pbArraySource:=IN_pbArraySource+1;
		OUT_wTargetWord14.8:=IN_pbArraySource^;
		IN_pbArraySource:=IN_pbArraySource+1;
		OUT_wTargetWord14.9:=IN_pbArraySource^;
		IN_pbArraySource:=IN_pbArraySource+1;
		OUT_wTargetWord14.10:=IN_pbArraySource^;
		IN_pbArraySource:=IN_pbArraySource+1;
		OUT_wTargetWord14.11:=IN_pbArraySource^;
		IN_pbArraySource:=IN_pbArraySource+1;
		OUT_wTargetWord14.12:=IN_pbArraySource^;
		IN_pbArraySource:=IN_pbArraySource+1;
		OUT_wTargetWord14.13:=IN_pbArraySource^;
		IN_pbArraySource:=IN_pbArraySource+1;
		OUT_wTargetWord14.14:=IN_pbArraySource^;
		IN_pbArraySource:=IN_pbArraySource+1;
		OUT_wTargetWord14.15:=IN_pbArraySource^;
		IN_pbArraySource:=IN_pbArraySource+1;
	END_IF	

(*******************************************************************************************************************************************)
(* Wort 15*)
(*******************************************************************************************************************************************)
(* Prüfen, ob Wort kopiert werden soll *)
	IF (IN_bCountWords >= 15) THEN
	(* Arraybereich kopieren *)
		OUT_wTargetWord15.0:=IN_pbArraySource^;
		IN_pbArraySource:=IN_pbArraySource+1;
		OUT_wTargetWord15.1:=IN_pbArraySource^;
		IN_pbArraySource:=IN_pbArraySource+1;
		OUT_wTargetWord15.2:=IN_pbArraySource^;
		IN_pbArraySource:=IN_pbArraySource+1;
		OUT_wTargetWord15.3:=IN_pbArraySource^;
		IN_pbArraySource:=IN_pbArraySource+1;
		OUT_wTargetWord15.4:=IN_pbArraySource^;
		IN_pbArraySource:=IN_pbArraySource+1;
		OUT_wTargetWord15.5:=IN_pbArraySource^;
		IN_pbArraySource:=IN_pbArraySource+1;
		OUT_wTargetWord15.6:=IN_pbArraySource^;
		IN_pbArraySource:=IN_pbArraySource+1;
		OUT_wTargetWord15.7:=IN_pbArraySource^;
		IN_pbArraySource:=IN_pbArraySource+1;
		OUT_wTargetWord15.8:=IN_pbArraySource^;
		IN_pbArraySource:=IN_pbArraySource+1;
		OUT_wTargetWord15.9:=IN_pbArraySource^;
		IN_pbArraySource:=IN_pbArraySource+1;
		OUT_wTargetWord15.10:=IN_pbArraySource^;
		IN_pbArraySource:=IN_pbArraySource+1;
		OUT_wTargetWord15.11:=IN_pbArraySource^;
		IN_pbArraySource:=IN_pbArraySource+1;
		OUT_wTargetWord15.12:=IN_pbArraySource^;
		IN_pbArraySource:=IN_pbArraySource+1;
		OUT_wTargetWord15.13:=IN_pbArraySource^;
		IN_pbArraySource:=IN_pbArraySource+1;
		OUT_wTargetWord15.14:=IN_pbArraySource^;
		IN_pbArraySource:=IN_pbArraySource+1;
		OUT_wTargetWord15.15:=IN_pbArraySource^;
		IN_pbArraySource:=IN_pbArraySource+1;
	END_IF	

